LIN {X 0,Y 310.323,Z 1135.59,A -85,B 0,C 180,E1 15003.805,E2 15003.805} C_VEL
LIN {X 0,Y 314.17,Z 1124.911,A -85,B 0,C 180,E1 14999.811,E2 14999.811} C_VEL
LIN {X 0,Y 318.874,Z 1112.724,A -85,B 0,C 180,E1 14996.072,E2 14996.072} C_VEL
LIN {X 0,Y 324.647,Z 1098.598,A -85,B 0,C 180,E1 14992.424,E2 14992.424} C_VEL
LIN {X 0,Y 330.405,Z 1084.681,A -85,B 0,C 180,E1 14989.411,E2 14989.411} C_VEL
LIN {X 0,Y 337.548,Z 1067.241,A -85,B 0,C 180,E1 14986.238,E2 14986.238} C_VEL
LIN {X 0,Y 344.264,Z 1050.446,A -85,B 0,C 180,E1 14983.682,E2 14983.682} C_VEL
LIN {X 0,Y 351.205,Z 1031.927,A -85,B 0,C 180,E1 14981.337,E2 14981.337} C_VEL
LIN {X 0,Y 357.94,Z 1012.865,A -85,B 0,C 180,E1 14979.306,E2 14979.306} C_VEL
LIN {X 0,Y 364.39,Z 992.442,A -85,B 0,C 180,E1 14977.528,E2 14977.528} C_VEL
LIN {X 0,Y 370.322,Z 971.659,A -85,B 0,C 180,E1 14976.036,E2 14976.036} C_VEL
LIN {X 0,Y 375.316,Z 951.31,A -85,B 0,C 180,E1 14974.861,E2 14974.861} C_VEL
LIN {X 0,Y 380.154,Z 927.978,A -85,B 0,C 180,E1 14973.796,E2 14973.796} C_VEL
LIN {X 0,Y 383.734,Z 906.313,A -85,B 0,C 180,E1 14973.058,E2 14973.058} C_VEL
LIN {X 0,Y 386.535,Z 881.758,A -85,B 0,C 180,E1 14972.438,E2 14972.438} C_VEL
LIN {X 0,Y 398.711,Z 690.492,A -85,B 0,C 180,E1 14968.671,E2 14968.671} C_VEL
LIN {X 0,Y 400.761,Z 658.99,A -85,B 0,C 180,E1 14968.053,E2 14968.053} C_VEL
LIN {X 0,Y 392.49,Z 644.745,A -85,B 0,C 180,E1 14965.137,E2 14965.137} C_VEL
LIN {X 0,Y 385.004,Z 632.908,A -85,B 0,C 180,E1 14962.121,E2 14962.121} C_VEL
LIN {X 0,Y 380.759,Z 626.867,A -85,B 0,C 180,E1 14960.2,E2 14960.2} C_VEL
LIN {X 0,Y 377.272,Z 622.196,A -85,B 0,C 180,E1 14958.463,E2 14958.463} C_VEL
LIN {X 0,Y 373.463,Z 617.117,A -85,B 0,C 180,E1 14956.326,E2 14956.326} C_VEL
LIN {X 0,Y 370.02,Z 612.377,A -85,B 0,C 180,E1 14954.075,E2 14954.075} C_VEL
LIN {X 0,Y 366.537,Z 608.515,A -85,B 0,C 180,E1 14951.406,E2 14951.406} C_VEL
LIN {X 0,Y 365.354,Z 606.34,A -85,B 0,C 180,E1 14950.246,E2 14950.246} C_VEL
LIN {X 0,Y 362.118,Z 603.229,A -85,B 0,C 180,E1 14946.5,E2 14946.5} C_VEL
LIN {X 0,Y 361.007,Z 600.343,A -85,B 0,C 180,E1 14944.129,E2 14944.129} C_VEL
LIN {X 0,Y 360.416,Z 600.177,A -85,B 0,C 180,E1 14936.819,E2 14936.819} C_VEL
LIN {X 0,Y 361.128,Z 600.593,A -85,B 0,C 180,E1 14934.996,E2 14934.996} C_VEL
LIN {X 0,Y 363.051,Z 604.515,A -85,B 0,C 180,E1 14931.607,E2 14931.607} C_VEL
LIN {X 0,Y 365.657,Z 606.777,A -85,B 0,C 180,E1 14928.885,E2 14928.885} C_VEL
LIN {X 0,Y 368.284,Z 610.838,A -85,B 0,C 180,E1 14926.577,E2 14926.577} C_VEL
LIN {X 0,Y 370.242,Z 612.802,A -85,B 0,C 180,E1 14925.187,E2 14925.187} C_VEL
LIN {X 0,Y 373.699,Z 617.381,A -85,B 0,C 180,E1 14922.964,E2 14922.964} C_VEL
LIN {X 0,Y 378.892,Z 624.313,A -85,B 0,C 180,E1 14920.138,E2 14920.138} C_VEL
LIN {X 0,Y 383.061,Z 630.072,A -85,B 0,C 180,E1 14918.164,E2 14918.164} C_VEL
LIN {X 0,Y 388.835,Z 638.03,A -85,B 0,C 180,E1 14915.746,E2 14915.746} C_VEL
LIN {X 0,Y 397.734,Z 651.353,A -85,B 0,C 180,E1 14912.488,E2 14912.488} C_VEL
LIN {X 0,Y 400.67,Z 656.231,A -85,B 0,C 180,E1 14911.501,E2 14911.501} C_VEL
LIN {X 0,Y 387.914,Z 856.221,A -85,B 0,C 180,E1 14907.587,E2 14907.587} C_VEL
LIN {X 0,Y 385.767,Z 879.846,A -85,B 0,C 180,E1 14907.046,E2 14907.046} C_VEL
LIN {X 0,Y 382.642,Z 902.799,A -85,B 0,C 180,E1 14906.324,E2 14906.324} C_VEL
LIN {X 0,Y 378.824,Z 923.719,A -85,B 0,C 180,E1 14905.436,E2 14905.436} C_VEL
LIN {X 0,Y 373.938,Z 945.868,A -85,B 0,C 180,E1 14904.246,E2 14904.246} C_VEL
LIN {X 0,Y 368.881,Z 965.062,A -85,B 0,C 180,E1 14902.964,E2 14902.964} C_VEL
LIN {X 0,Y 362.451,Z 986.567,A -85,B 0,C 180,E1 14901.211,E2 14901.211} C_VEL
LIN {X 0,Y 356.513,Z 1004.243,A -85,B 0,C 180,E1 14899.468,E2 14899.468} C_VEL
LIN {X 0,Y 349.249,Z 1023.997,A -85,B 0,C 180,E1 14897.131,E2 14897.131} C_VEL
LIN {X 0,Y 342.731,Z 1040.527,A -85,B 0,C 180,E1 14894.793,E2 14894.793} C_VEL
LIN {X 0,Y 335.925,Z 1056.776,A -85,B 0,C 180,E1 14892.045,E2 14892.045} C_VEL
LIN {X 0,Y 329.503,Z 1071.829,A -85,B 0,C 180,E1 14889.029,E2 14889.029} C_VEL
LIN {X 0,Y 323.5,Z 1085.447,A -85,B 0,C 180,E1 14885.744,E2 14885.744} C_VEL
LIN {X 0,Y 318.06,Z 1098.198,A -85,B 0,C 180,E1 14882.092,E2 14882.092} C_VEL
LIN {X 0,Y 313.614,Z 1108.925,A -85,B 0,C 180,E1 14878.363,E2 14878.363} C_VEL
LIN {X 0,Y 309.706,Z 1119.272,A -85,B 0,C 180,E1 14873.986,E2 14873.986} C_VEL
LIN {X 0,Y 307.195,Z 1126.919,A -85,B 0,C 180,E1 14869.984,E2 14869.984} C_VEL
LIN {X 0,Y 305.468,Z 1133.25,A -85,B 0,C 180,E1 14865.765,E2 14865.765} C_VEL
LIN {X 0,Y 304.592,Z 1137.667,A -85,B 0,C 180,E1 14861.936,E2 14861.936} C_VEL
LIN {X 0,Y 304.117,Z 1141.074,A -85,B 0,C 180,E1 14857.747,E2 14857.747} C_VEL
LIN {X 0,Y 303.996,Z 1142.818,A -85,B 0,C 180,E1 14854.15,E2 14854.15} C_VEL
LIN {X 0,Y 303.963,Z 1143.581,A -85,B 0,C 180,E1 14850.326,E2 14850.326} C_VEL
LIN {X 0,Y 303.98,Z 1142.983,A -85,B 0,C 180,E1 14846.229,E2 14846.229} C_VEL
LIN {X 0,Y 304.085,Z 1141.349,A -85,B 0,C 180,E1 14842.633,E2 14842.633} C_VEL
LIN {X 0,Y 304.486,Z 1138.367,A -85,B 0,C 180,E1 14838.637,E2 14838.637} C_VEL
LIN {X 0,Y 305.382,Z 1133.619,A -85,B 0,C 180,E1 14834.427,E2 14834.427} C_VEL
LIN {X 0,Y 305.467,Z 1133.26,A -85,B 0,C 180,E1 14834.147,E2 14834.147} C_VEL
LIN {X 0,Y 304.971,Z 1131.474,A -85,B 0,C 180,E1 14832.733,E2 14832.733} C_VEL
LIN {X 0,Y 300.512,Z 1126.313,A -85,B 0,C 180,E1 14828.918,E2 14828.918} C_VEL
LIN {X 0,Y 300.483,Z 1124.298,A -85,B 0,C 180,E1 14827.7,E2 14827.7} C_VEL
LIN {X 0,Y 303.77,Z 1115.533,A -85,B 0,C 180,E1 14823.408,E2 14823.408} C_VEL
LIN {X 0,Y 307.804,Z 1105.953,A -85,B 0,C 180,E1 14819.553,E2 14819.553} C_VEL
LIN {X 0,Y 312.855,Z 1094.529,A -85,B 0,C 180,E1 14815.773,E2 14815.773} C_VEL
LIN {X 0,Y 318.735,Z 1081.794,A -85,B 0,C 180,E1 14812.234,E2 14812.234} C_VEL
LIN {X 0,Y 325.377,Z 1067.137,A -85,B 0,C 180,E1 14808.883,E2 14808.883} C_VEL
LIN {X 0,Y 332.647,Z 1050.932,A -85,B 0,C 180,E1 14805.786,E2 14805.786} C_VEL
LIN {X 0,Y 339.306,Z 1035.304,A -85,B 0,C 180,E1 14803.293,E2 14803.293} C_VEL
LIN {X 0,Y 347.012,Z 1016.058,A -85,B 0,C 180,E1 14800.73,E2 14800.73} C_VEL
LIN {X 0,Y 353.723,Z 997.925,A -85,B 0,C 180,E1 14798.725,E2 14798.725} C_VEL
LIN {X 0,Y 360.235,Z 978.29,A -85,B 0,C 180,E1 14796.931,E2 14796.931} C_VEL
LIN {X 0,Y 366.199,Z 958.243,A -85,B 0,C 180,E1 14795.411,E2 14795.411} C_VEL
LIN {X 0,Y 371.457,Z 937.38,A -85,B 0,C 180,E1 14794.136,E2 14794.136} C_VEL
LIN {X 0,Y 376.2,Z 915.233,A -85,B 0,C 180,E1 14793.049,E2 14793.049} C_VEL
LIN {X 0,Y 379.82,Z 893.219,A -85,B 0,C 180,E1 14792.229,E2 14792.229} C_VEL
LIN {X 0,Y 382.736,Z 869.272,A -85,B 0,C 180,E1 14791.578,E2 14791.578} C_VEL
LIN {X 0,Y 394.662,Z 690.82,A -85,B 0,C 180,E1 14788.052,E2 14788.052} C_VEL
LIN {X 0,Y 396.631,Z 660.49,A -85,B 0,C 180,E1 14787.432,E2 14787.432} C_VEL
LIN {X 0,Y 388.655,Z 648.175,A -85,B 0,C 180,E1 14784.509,E2 14784.509} C_VEL
LIN {X 0,Y 382.448,Z 639.194,A -85,B 0,C 180,E1 14781.913,E2 14781.913} C_VEL
LIN {X 0,Y 378.405,Z 633.571,A -85,B 0,C 180,E1 14780.01,E2 14780.01} C_VEL
LIN {X 0,Y 375.594,Z 629.676,A -85,B 0,C 180,E1 14778.549,E2 14778.549} C_VEL
LIN {X 0,Y 371.88,Z 624.709,A -85,B 0,C 180,E1 14776.398,E2 14776.398} C_VEL
LIN {X 0,Y 368.336,Z 619.786,A -85,B 0,C 180,E1 14773.981,E2 14773.981} C_VEL
LIN {X 0,Y 365.292,Z 616.25,A -85,B 0,C 180,E1 14771.526,E2 14771.526} C_VEL
LIN {X 0,Y 364.226,Z 614.277,A -85,B 0,C 180,E1 14770.439,E2 14770.439} C_VEL
LIN {X 0,Y 361.038,Z 611.018,A -85,B 0,C 180,E1 14766.52,E2 14766.52} C_VEL
LIN {X 0,Y 360.042,Z 608.276,A -85,B 0,C 180,E1 14764.141,E2 14764.141} C_VEL
LIN {X 0,Y 360.043,Z 608.283,A -85,B 0,C 180,E1 14756.338,E2 14756.338} C_VEL
LIN {X 0,Y 362.332,Z 612.803,A -85,B 0,C 180,E1 14752.07,E2 14752.07} C_VEL
LIN {X 0,Y 364.46,Z 614.581,A -85,B 0,C 180,E1 14749.808,E2 14749.808} C_VEL
LIN {X 0,Y 367.19,Z 618.789,A -85,B 0,C 180,E1 14747.338,E2 14747.338} C_VEL
LIN {X 0,Y 368.856,Z 620.49,A -85,B 0,C 180,E1 14746.12,E2 14746.12} C_VEL
LIN {X 0,Y 372.39,Z 625.157,A -85,B 0,C 180,E1 14743.786,E2 14743.786} C_VEL
LIN {X 0,Y 377.467,Z 632.272,A -85,B 0,C 180,E1 14740.946,E2 14740.946} C_VEL
LIN {X 0,Y 381.184,Z 637.463,A -85,B 0,C 180,E1 14739.141,E2 14739.141} C_VEL
LIN {X 0,Y 385.902,Z 644.86,A -85,B 0,C 180,E1 14737.05,E2 14737.05} C_VEL
LIN {X 0,Y 391.999,Z 654.977,A -85,B 0,C 180,E1 14734.627,E2 14734.627} C_VEL
LIN {X 0,Y 396.821,Z 663.696,A -85,B 0,C 180,E1 14732.874,E2 14732.874} C_VEL
LIN {X 0,Y 382.995,Z 873.743,A -85,B 0,C 180,E1 14728.753,E2 14728.753} C_VEL
LIN {X 0,Y 380.728,Z 896.852,A -85,B 0,C 180,E1 14728.218,E2 14728.218} C_VEL
LIN {X 0,Y 376.911,Z 921.624,A -85,B 0,C 180,E1 14727.459,E2 14727.459} C_VEL
LIN {X 0,Y 372.941,Z 941.713,A -85,B 0,C 180,E1 14726.63,E2 14726.63} C_VEL
LIN {X 0,Y 367.489,Z 964.391,A -85,B 0,C 180,E1 14725.43,E2 14725.43} C_VEL
LIN {X 0,Y 361.774,Z 984.881,A -85,B 0,C 180,E1 14724.075,E2 14724.075} C_VEL
LIN {X 0,Y 355.238,Z 1005.335,A -85,B 0,C 180,E1 14722.402,E2 14722.402} C_VEL
LIN {X 0,Y 348.52,Z 1024.568,A -85,B 0,C 180,E1 14720.509,E2 14720.509} C_VEL
LIN {X 0,Y 341.201,Z 1043.572,A -85,B 0,C 180,E1 14718.227,E2 14718.227} C_VEL
LIN {X 0,Y 333.849,Z 1061.702,A -85,B 0,C 180,E1 14715.622,E2 14715.622} C_VEL
LIN {X 0,Y 327.017,Z 1077.671,A -85,B 0,C 180,E1 14712.867,E2 14712.867} C_VEL
LIN {X 0,Y 319.73,Z 1094.407,A -85,B 0,C 180,E1 14709.406,E2 14709.406} C_VEL
LIN {X 0,Y 313.658,Z 1108.501,A -85,B 0,C 180,E1 14705.912,E2 14705.912} C_VEL
LIN {X 0,Y 308.33,Z 1121.103,A -85,B 0,C 180,E1 14702.128,E2 14702.128} C_VEL
LIN {X 0,Y 303.91,Z 1132.469,A -85,B 0,C 180,E1 14698.064,E2 14698.064} C_VEL
LIN {X 0,Y 300.611,Z 1141.876,A -85,B 0,C 180,E1 14693.94,E2 14693.94} C_VEL
LIN {X 0,Y 298.166,Z 1150.31,A -85,B 0,C 180,E1 14689.389,E2 14689.389} C_VEL
LIN {X 0,Y 296.881,Z 1156.088,A -85,B 0,C 180,E1 14685.43,E2 14685.43} C_VEL
LIN {X 0,Y 296.169,Z 1161.086,A -85,B 0,C 180,E1 14680.897,E2 14680.897} C_VEL
LIN {X 0,Y 295.965,Z 1163.871,A -85,B 0,C 180,E1 14677.18,E2 14677.18} C_VEL
LIN {X 0,Y 295.95,Z 1165.555,A -85,B 0,C 180,E1 14673.486,E2 14673.486} C_VEL
LIN {X 0,Y 295.962,Z 1166.074,A -85,B 0,C 180,E1 14669.59,E2 14669.59} C_VEL
LIN {X 0,Y 295.962,Z 1165.342,A -85,B 0,C 180,E1 14665.931,E2 14665.931} C_VEL
LIN {X 0,Y 295.992,Z 1163.512,A -85,B 0,C 180,E1 14662.234,E2 14662.234} C_VEL
LIN {X 0,Y 296.296,Z 1159.96,A -85,B 0,C 180,E1 14657.923,E2 14657.923} C_VEL
LIN {X 0,Y 297.034,Z 1155.291,A -85,B 0,C 180,E1 14653.976,E2 14653.976} C_VEL
LIN {X 0,Y 298.61,Z 1148.673,A -85,B 0,C 180,E1 14649.62,E2 14649.62} C_VEL
LIN {X 0,Y 301.021,Z 1140.61,A -85,B 0,C 180,E1 14645.468,E2 14645.468} C_VEL
LIN {X 0,Y 304.663,Z 1130.418,A -85,B 0,C 180,E1 14641.155,E2 14641.155} C_VEL
LIN {X 0,Y 309.058,Z 1119.318,A -85,B 0,C 180,E1 14637.297,E2 14637.297} C_VEL
LIN {X 0,Y 314.85,Z 1105.605,A -85,B 0,C 180,E1 14633.342,E2 14633.342} C_VEL
LIN {X 0,Y 321.144,Z 1091.219,A -85,B 0,C 180,E1 14629.872,E2 14629.872} C_VEL
LIN {X 0,Y 328.027,Z 1075.258,A -85,B 0,C 180,E1 14626.699,E2 14626.699} C_VEL
LIN {X 0,Y 335.328,Z 1058.003,A -85,B 0,C 180,E1 14623.814,E2 14623.814} C_VEL
LIN {X 0,Y 342.149,Z 1041.054,A -85,B 0,C 180,E1 14621.455,E2 14621.455} C_VEL
LIN {X 0,Y 349.556,Z 1021.471,A -85,B 0,C 180,E1 14619.179,E2 14619.179} C_VEL
LIN {X 0,Y 356.069,Z 1002.737,A -85,B 0,C 180,E1 14617.374,E2 14617.374} C_VEL
LIN {X 0,Y 362.647,Z 981.642,A -85,B 0,C 180,E1 14615.706,E2 14615.706} C_VEL
LIN {X 0,Y 368.003,Z 962.244,A -85,B 0,C 180,E1 14614.45,E2 14614.45} C_VEL
LIN {X 0,Y 373.241,Z 939.947,A -85,B 0,C 180,E1 14613.299,E2 14613.299} C_VEL
LIN {X 0,Y 377.27,Z 919.347,A -85,B 0,C 180,E1 14612.467,E2 14612.467} C_VEL
LIN {X 0,Y 380.769,Z 895.853,A -85,B 0,C 180,E1 14611.764,E2 14611.764} C_VEL
LIN {X 0,Y 383.036,Z 872.053,A -85,B 0,C 180,E1 14611.22,E2 14611.22} C_VEL
LIN {X 0,Y 396.739,Z 663.465,A -85,B 0,C 180,E1 14607.129,E2 14607.129} C_VEL
LIN {X 0,Y 389.401,Z 650.607,A -85,B 0,C 180,E1 14604.418,E2 14604.418} C_VEL
LIN {X 0,Y 382.164,Z 638.896,A -85,B 0,C 180,E1 14601.365,E2 14601.365} C_VEL
LIN {X 0,Y 378.422,Z 633.662,A -85,B 0,C 180,E1 14599.606,E2 14599.606} C_VEL
LIN {X 0,Y 375.456,Z 629.581,A -85,B 0,C 180,E1 14598.074,E2 14598.074} C_VEL
LIN {X 0,Y 371.864,Z 624.679,A -85,B 0,C 180,E1 14595.997,E2 14595.997} C_VEL
LIN {X 0,Y 368.174,Z 619.697,A -85,B 0,C 180,E1 14593.506,E2 14593.506} C_VEL
LIN {X 0,Y 365.049,Z 615.916,A -85,B 0,C 180,E1 14590.973,E2 14590.973} C_VEL
LIN {X 0,Y 364.052,Z 614.127,A -85,B 0,C 180,E1 14589.963,E2 14589.963} C_VEL
LIN {X 0,Y 360.855,Z 610.766,A -85,B 0,C 180,E1 14586.044,E2 14586.044} C_VEL
LIN {X 0,Y 359.96,Z 608.269,A -85,B 0,C 180,E1 14583.982,E2 14583.982} C_VEL
LIN {X 0,Y 359.498,Z 608.138,A -85,B 0,C 180,E1 14576.633,E2 14576.633} C_VEL
LIN {X 0,Y 360.078,Z 608.513,A -85,B 0,C 180,E1 14575.141,E2 14575.141} C_VEL
LIN {X 0,Y 361.954,Z 612.395,A -85,B 0,C 180,E1 14571.741,E2 14571.741} C_VEL
LIN {X 0,Y 364.428,Z 614.657,A -85,B 0,C 180,E1 14569.087,E2 14569.087} C_VEL
LIN {X 0,Y 367.013,Z 618.639,A -85,B 0,C 180,E1 14566.771,E2 14566.771} C_VEL
LIN {X 0,Y 368.791,Z 620.478,A -85,B 0,C 180,E1 14565.476,E2 14565.476} C_VEL
LIN {X 0,Y 372.223,Z 625.071,A -85,B 0,C 180,E1 14563.216,E2 14563.216} C_VEL
LIN {X 0,Y 377.185,Z 631.895,A -85,B 0,C 180,E1 14560.447,E2 14560.447} C_VEL
LIN {X 0,Y 381.204,Z 637.558,A -85,B 0,C 180,E1 14558.497,E2 14558.497} C_VEL
LIN {X 0,Y 386.708,Z 645.323,A -85,B 0,C 180,E1 14556.131,E2 14556.131} C_VEL
LIN {X 0,Y 395.16,Z 658.231,A -85,B 0,C 180,E1 14552.95,E2 14552.95} C_VEL
LIN {X 0,Y 396.616,Z 660.877,A -85,B 0,C 180,E1 14552.433,E2 14552.433} C_VEL
LIN {X 0,Y 383.418,Z 860.114,A -85,B 0,C 180,E1 14548.521,E2 14548.521} C_VEL
LIN {X 0,Y 381.23,Z 882.282,A -85,B 0,C 180,E1 14547.997,E2 14547.997} C_VEL
LIN {X 0,Y 377.759,Z 905.918,A -85,B 0,C 180,E1 14547.224,E2 14547.224} C_VEL
LIN {X 0,Y 373.897,Z 926.162,A -85,B 0,C 180,E1 14546.347,E2 14546.347} C_VEL
LIN {X 0,Y 368.699,Z 948.424,A -85,B 0,C 180,E1 14545.119,E2 14545.119} C_VEL
LIN {X 0,Y 363.509,Z 967.365,A -85,B 0,C 180,E1 14543.833,E2 14543.833} C_VEL
LIN {X 0,Y 357.121,Z 987.761,A -85,B 0,C 180,E1 14542.143,E2 14542.143} C_VEL
LIN {X 0,Y 350.732,Z 1006.09,A -85,B 0,C 180,E1 14540.314,E2 14540.314} C_VEL
LIN {X 0,Y 343.482,Z 1024.939,A -85,B 0,C 180,E1 14538.046,E2 14538.046} C_VEL
LIN {X 0,Y 336.512,Z 1041.934,A -85,B 0,C 180,E1 14535.61,E2 14535.61} C_VEL
LIN {X 0,Y 329.446,Z 1058,A -85,B 0,C 180,E1 14532.832,E2 14532.832} C_VEL
LIN {X 0,Y 322.577,Z 1073.326,A -85,B 0,C 180,E1 14529.682,E2 14529.682} C_VEL
LIN {X 0,Y 316.51,Z 1086.447,A -85,B 0,C 180,E1 14526.435,E2 14526.435} C_VEL
LIN {X 0,Y 310.555,Z 1099.631,A -85,B 0,C 180,E1 14522.526,E2 14522.526} C_VEL
LIN {X 0,Y 306.154,Z 1109.739,A -85,B 0,C 180,E1 14518.905,E2 14518.905} C_VEL
LIN {X 0,Y 302.201,Z 1119.55,A -85,B 0,C 180,E1 14514.639,E2 14514.639} C_VEL
LIN {X 0,Y 299.495,Z 1127.228,A -85,B 0,C 180,E1 14510.521,E2 14510.521} C_VEL
LIN {X 0,Y 297.582,Z 1133.714,A -85,B 0,C 180,E1 14506.065,E2 14506.065} C_VEL
LIN {X 0,Y 296.599,Z 1138.371,A -85,B 0,C 180,E1 14501.867,E2 14501.867} C_VEL
LIN {X 0,Y 296.112,Z 1141.595,A -85,B 0,C 180,E1 14497.568,E2 14497.568} C_VEL
LIN {X 0,Y 295.995,Z 1143.249,A -85,B 0,C 180,E1 14493.874,E2 14493.874} C_VEL
LIN {X 0,Y 295.973,Z 1143.908,A -85,B 0,C 180,E1 14489.807,E2 14489.807} C_VEL
LIN {X 0,Y 296.002,Z 1143.152,A -85,B 0,C 180,E1 14485.739,E2 14485.739} C_VEL
LIN {X 0,Y 296.158,Z 1141.323,A -85,B 0,C 180,E1 14481.849,E2 14481.849} C_VEL
LIN {X 0,Y 296.71,Z 1137.672,A -85,B 0,C 180,E1 14477.348,E2 14477.348} C_VEL
LIN {X 0,Y 297.806,Z 1132.941,A -85,B 0,C 180,E1 14473.218,E2 14473.218} C_VEL
LIN {X 0,Y 299.892,Z 1126.025,A -85,B 0,C 180,E1 14468.69,E2 14468.69} C_VEL
LIN {X 0,Y 300.483,Z 1124.298,A -85,B 0,C 180,E1 14467.7,E2 14467.7} C_VEL
LIN {X 0,Y 300.434,Z 1121.89,A -85,B 0,C 180,E1 14466.293,E2 14466.293} C_VEL
LIN {X 0,Y 297.378,Z 1115.16,A -85,B 0,C 180,E1 14462.471,E2 14462.471} C_VEL
LIN {X 0,Y 297.827,Z 1112.655,A -85,B 0,C 180,E1 14461.283,E2 14461.283} C_VEL
LIN {X 0,Y 302.7,Z 1101.884,A -85,B 0,C 180,E1 14457.2,E2 14457.2} C_VEL
LIN {X 0,Y 308.496,Z 1089.823,A -85,B 0,C 180,E1 14453.391,E2 14453.391} C_VEL
LIN {X 0,Y 315.005,Z 1076.254,A -85,B 0,C 180,E1 14449.884,E2 14449.884} C_VEL
LIN {X 0,Y 322.472,Z 1060.543,A -85,B 0,C 180,E1 14446.502,E2 14446.502} C_VEL
LIN {X 0,Y 329.497,Z 1045.241,A -85,B 0,C 180,E1 14443.763,E2 14443.763} C_VEL
LIN {X 0,Y 337.167,Z 1027.551,A -85,B 0,C 180,E1 14441.129,E2 14441.129} C_VEL
LIN {X 0,Y 344.124,Z 1010.415,A -85,B 0,C 180,E1 14438.993,E2 14438.993} C_VEL
LIN {X 0,Y 351.191,Z 991.173,A -85,B 0,C 180,E1 14437.004,E2 14437.004} C_VEL
LIN {X 0,Y 357.477,Z 972.322,A -85,B 0,C 180,E1 14435.379,E2 14435.379} C_VEL
LIN {X 0,Y 363.46,Z 951.595,A -85,B 0,C 180,E1 14433.921,E2 14433.921} C_VEL
LIN {X 0,Y 368.561,Z 931.288,A -85,B 0,C 180,E1 14432.755,E2 14432.755} C_VEL
LIN {X 0,Y 372.973,Z 909.487,A -85,B 0,C 180,E1 14431.773,E2 14431.773} C_VEL
LIN {X 0,Y 376.463,Z 888.081,A -85,B 0,C 180,E1 14431.026,E2 14431.026} C_VEL
LIN {X 0,Y 378.998,Z 864.998,A -85,B 0,C 180,E1 14430.448,E2 14430.448} C_VEL
LIN {X 0,Y 392.66,Z 667.126,A -85,B 0,C 180,E1 14426.551,E2 14426.551} C_VEL
LIN {X 0,Y 392.75,Z 665.236,A -85,B 0,C 180,E1 14426.501,E2 14426.501} C_VEL
LIN {X 0,Y 384.149,Z 651.782,A -85,B 0,C 180,E1 14423.143,E2 14423.143} C_VEL
LIN {X 0,Y 377.425,Z 642.064,A -85,B 0,C 180,E1 14420.064,E2 14420.064} C_VEL
LIN {X 0,Y 373.665,Z 636.906,A -85,B 0,C 180,E1 14418.083,E2 14418.083} C_VEL
LIN {X 0,Y 370.3,Z 632.269,A -85,B 0,C 180,E1 14416.067,E2 14416.067} C_VEL
LIN {X 0,Y 366.734,Z 627.329,A -85,B 0,C 180,E1 14413.561,E2 14413.561} C_VEL
LIN {X 0,Y 363.749,Z 623.51,A -85,B 0,C 180,E1 14411.014,E2 14411.014} C_VEL
LIN {X 0,Y 362.935,Z 622.069,A -85,B 0,C 180,E1 14410.156,E2 14410.156} C_VEL
LIN {X 0,Y 359.883,Z 618.731,A -85,B 0,C 180,E1 14406.221,E2 14406.221} C_VEL
LIN {X 0,Y 359.005,Z 616.202,A -85,B 0,C 180,E1 14403.993,E2 14403.993} C_VEL
LIN {X 0,Y 359.07,Z 616.224,A -85,B 0,C 180,E1 14396.328,E2 14396.328} C_VEL
LIN {X 0,Y 360.991,Z 620.417,A -85,B 0,C 180,E1 14392.52,E2 14392.52} C_VEL
LIN {X 0,Y 363.241,Z 622.444,A -85,B 0,C 180,E1 14390.014,E2 14390.014} C_VEL
LIN {X 0,Y 365.923,Z 626.589,A -85,B 0,C 180,E1 14387.534,E2 14387.534} C_VEL
LIN {X 0,Y 367.549,Z 628.4,A -85,B 0,C 180,E1 14386.31,E2 14386.31} C_VEL
LIN {X 0,Y 371.506,Z 633.867,A -85,B 0,C 180,E1 14383.666,E2 14383.666} C_VEL
LIN {X 0,Y 375.63,Z 639.633,A -85,B 0,C 180,E1 14381.332,E2 14381.332} C_VEL
LIN {X 0,Y 379.571,Z 645.276,A -85,B 0,C 180,E1 14379.371,E2 14379.371} C_VEL
LIN {X 0,Y 384.969,Z 653.991,A -85,B 0,C 180,E1 14376.95,E2 14376.95} C_VEL
LIN {X 0,Y 391.59,Z 665.539,A -85,B 0,C 180,E1 14374.315,E2 14374.315} C_VEL
LIN {X 0,Y 392.874,Z 668.184,A -85,B 0,C 180,E1 14373.826,E2 14373.826} C_VEL
LIN {X 0,Y 378.717,Z 875.394,A -85,B 0,C 180,E1 14369.752,E2 14369.752} C_VEL
LIN {X 0,Y 376.41,Z 897.705,A -85,B 0,C 180,E1 14369.23,E2 14369.23} C_VEL
LIN {X 0,Y 372.481,Z 922.139,A -85,B 0,C 180,E1 14368.475,E2 14368.475} C_VEL
LIN {X 0,Y 368.231,Z 942.906,A -85,B 0,C 180,E1 14367.614,E2 14367.614} C_VEL
LIN {X 0,Y 362.847,Z 964.426,A -85,B 0,C 180,E1 14366.467,E2 14366.467} C_VEL
LIN {X 0,Y 357.046,Z 984.581,A -85,B 0,C 180,E1 14365.136,E2 14365.136} C_VEL
LIN {X 0,Y 350.214,Z 1005.252,A -85,B 0,C 180,E1 14363.446,E2 14363.446} C_VEL
LIN {X 0,Y 343.072,Z 1024.958,A -85,B 0,C 180,E1 14361.497,E2 14361.497} C_VEL
LIN {X 0,Y 335.478,Z 1043.88,A -85,B 0,C 180,E1 14359.202,E2 14359.202} C_VEL
LIN {X 0,Y 327.54,Z 1062.576,A -85,B 0,C 180,E1 14356.469,E2 14356.469} C_VEL
LIN {X 0,Y 320.526,Z 1078.3,A -85,B 0,C 180,E1 14353.705,E2 14353.705} C_VEL
LIN {X 0,Y 313.292,Z 1094.094,A -85,B 0,C 180,E1 14350.381,E2 14350.381} C_VEL
LIN {X 0,Y 306.905,Z 1108.188,A -85,B 0,C 180,E1 14346.83,E2 14346.83} C_VEL
LIN {X 0,Y 301.256,Z 1120.79,A -85,B 0,C 180,E1 14342.977,E2 14342.977} C_VEL
LIN {X 0,Y 296.551,Z 1132.156,A -85,B 0,C 180,E1 14338.825,E2 14338.825} C_VEL
LIN {X 0,Y 293.017,Z 1141.565,A -85,B 0,C 180,E1 14334.601,E2 14334.601} C_VEL
LIN {X 0,Y 290.379,Z 1150.001,A -85,B 0,C 180,E1 14329.93,E2 14329.93} C_VEL
LIN {X 0,Y 288.981,Z 1155.781,A -85,B 0,C 180,E1 14325.862,E2 14325.862} C_VEL
LIN {X 0,Y 288.202,Z 1160.782,A -85,B 0,C 180,E1 14321.202,E2 14321.202} C_VEL
LIN {X 0,Y 287.97,Z 1163.569,A -85,B 0,C 180,E1 14317.381,E2 14317.381} C_VEL
LIN {X 0,Y 287.956,Z 1165.255,A -85,B 0,C 180,E1 14313.583,E2 14313.583} C_VEL
LIN {X 0,Y 287.966,Z 1165.766,A -85,B 0,C 180,E1 14309.509,E2 14309.509} C_VEL
LIN {X 0,Y 287.966,Z 1164.97,A -85,B 0,C 180,E1 14305.619,E2 14305.619} C_VEL
LIN {X 0,Y 288.021,Z 1163.091,A -85,B 0,C 180,E1 14301.817,E2 14301.817} C_VEL
LIN {X 0,Y 288.364,Z 1159.441,A -85,B 0,C 180,E1 14297.382,E2 14297.382} C_VEL
LIN {X 0,Y 289.228,Z 1154.624,A -85,B 0,C 180,E1 14293.251,E2 14293.251} C_VEL
LIN {X 0,Y 291.159,Z 1147.27,A -85,B 0,C 180,E1 14288.441,E2 14288.441} C_VEL
LIN {X 0,Y 293.755,Z 1139.463,A -85,B 0,C 180,E1 14284.388,E2 14284.388} C_VEL
LIN {X 0,Y 297.766,Z 1129.048,A -85,B 0,C 180,E1 14279.978,E2 14279.978} C_VEL
LIN {X 0,Y 302.582,Z 1117.795,A -85,B 0,C 180,E1 14276.037,E2 14276.037} C_VEL
LIN {X 0,Y 308.469,Z 1104.573,A -85,B 0,C 180,E1 14272.22,E2 14272.22} C_VEL
LIN {X 0,Y 315.161,Z 1090.063,A -85,B 0,C 180,E1 14268.708,E2 14268.708} C_VEL
LIN {X 0,Y 322.204,Z 1074.472,A -85,B 0,C 180,E1 14265.591,E2 14265.591} C_VEL
LIN {X 0,Y 330.086,Z 1056.563,A -85,B 0,C 180,E1 14262.602,E2 14262.602} C_VEL
LIN {X 0,Y 337.079,Z 1039.888,A -85,B 0,C 180,E1 14260.288,E2 14260.288} C_VEL
LIN {X 0,Y 344.682,Z 1020.416,A -85,B 0,C 180,E1 14258.04,E2 14258.04} C_VEL
LIN {X 0,Y 351.152,Z 1002.425,A -85,B 0,C 180,E1 14256.311,E2 14256.311} C_VEL
LIN {X 0,Y 357.935,Z 981.358,A -85,B 0,C 180,E1 14254.647,E2 14254.647} C_VEL
LIN {X 0,Y 363.604,Z 961.44,A -85,B 0,C 180,E1 14253.364,E2 14253.364} C_VEL
LIN {X 0,Y 368.859,Z 939.635,A -85,B 0,C 180,E1 14252.248,E2 14252.248} C_VEL
LIN {X 0,Y 372.94,Z 919.361,A -85,B 0,C 180,E1 14251.434,E2 14251.434} C_VEL
LIN {X 0,Y 376.574,Z 895.699,A -85,B 0,C 180,E1 14250.727,E2 14250.727} C_VEL
LIN {X 0,Y 378.909,Z 871.983,A -85,B 0,C 180,E1 14250.184,E2 14250.184} C_VEL
LIN {X 0,Y 392.788,Z 667.957,A -85,B 0,C 180,E1 14246.177,E2 14246.177} C_VEL
LIN {X 0,Y 386.541,Z 656.796,A -85,B 0,C 180,E1 14243.758,E2 14243.758} C_VEL
LIN {X 0,Y 379.99,Z 645.93,A -85,B 0,C 180,E1 14240.887,E2 14240.887} C_VEL
LIN {X 0,Y 376.129,Z 640.435,A -85,B 0,C 180,E1 14239.004,E2 14239.004} C_VEL
LIN {X 0,Y 373.523,Z 636.805,A -85,B 0,C 180,E1 14237.606,E2 14237.606} C_VEL
LIN {X 0,Y 370.155,Z 632.107,A -85,B 0,C 180,E1 14235.591,E2 14235.591} C_VEL
LIN {X 0,Y 366.781,Z 627.408,A -85,B 0,C 180,E1 14233.237,E2 14233.237} C_VEL
LIN {X 0,Y 363.659,Z 623.461,A -85,B 0,C 180,E1 14230.615,E2 14230.615} C_VEL
LIN {X 0,Y 362.76,Z 621.909,A -85,B 0,C 180,E1 14229.679,E2 14229.679} C_VEL
LIN {X 0,Y 359.699,Z 618.474,A -85,B 0,C 180,E1 14225.743,E2 14225.743} C_VEL
LIN {X 0,Y 358.916,Z 616.194,A -85,B 0,C 180,E1 14223.833,E2 14223.833} C_VEL
LIN {X 0,Y 358.524,Z 616.079,A -85,B 0,C 180,E1 14216.625,E2 14216.625} C_VEL
LIN {X 0,Y 359.031,Z 616.429,A -85,B 0,C 180,E1 14215.287,E2 14215.287} C_VEL
LIN {X 0,Y 360.859,Z 620.274,A -85,B 0,C 180,E1 14211.876,E2 14211.876} C_VEL
LIN {X 0,Y 363.134,Z 622.366,A -85,B 0,C 180,E1 14209.369,E2 14209.369} C_VEL
LIN {X 0,Y 365.846,Z 626.54,A -85,B 0,C 180,E1 14206.889,E2 14206.889} C_VEL
LIN {X 0,Y 367.384,Z 628.213,A -85,B 0,C 180,E1 14205.741,E2 14205.741} C_VEL
LIN {X 0,Y 371.592,Z 634.097,A -85,B 0,C 180,E1 14202.945,E2 14202.945} C_VEL
LIN {X 0,Y 375.489,Z 639.472,A -85,B 0,C 180,E1 14200.76,E2 14200.76} C_VEL
LIN {X 0,Y 379.437,Z 645.153,A -85,B 0,C 180,E1 14198.797,E2 14198.797} C_VEL
LIN {X 0,Y 384.848,Z 653.017,A -85,B 0,C 180,E1 14196.415,E2 14196.415} C_VEL
LIN {X 0,Y 392.684,Z 665.231,A -85,B 0,C 180,E1 14193.391,E2 14193.391} C_VEL
LIN {X 0,Y 379.342,Z 859.968,A -85,B 0,C 180,E1 14189.562,E2 14189.562} C_VEL
LIN {X 0,Y 377.083,Z 882.308,A -85,B 0,C 180,E1 14189.036,E2 14189.036} C_VEL
LIN {X 0,Y 373.477,Z 906.23,A -85,B 0,C 180,E1 14188.258,E2 14188.258} C_VEL
LIN {X 0,Y 369.546,Z 926.262,A -85,B 0,C 180,E1 14187.395,E2 14187.395} C_VEL
LIN {X 0,Y 364.118,Z 948.845,A -85,B 0,C 180,E1 14186.153,E2 14186.153} C_VEL
LIN {X 0,Y 358.508,Z 968.672,A -85,B 0,C 180,E1 14184.803,E2 14184.803} C_VEL
LIN {X 0,Y 351.917,Z 988.875,A -85,B 0,C 180,E1 14183.111,E2 14183.111} C_VEL
LIN {X 0,Y 345.09,Z 1007.772,A -85,B 0,C 180,E1 14181.206,E2 14181.206} C_VEL
LIN {X 0,Y 337.832,Z 1025.82,A -85,B 0,C 180,E1 14179.001,E2 14179.001} C_VEL
LIN {X 0,Y 330.595,Z 1042.787,A -85,B 0,C 180,E1 14176.541,E2 14176.541} C_VEL
LIN {X 0,Y 323.032,Z 1059.224,A -85,B 0,C 180,E1 14173.65,E2 14173.65} C_VEL
LIN {X 0,Y 315.884,Z 1074.396,A -85,B 0,C 180,E1 14170.458,E2 14170.458} C_VEL
LIN {X 0,Y 309.569,Z 1087.447,A -85,B 0,C 180,E1 14167.156,E2 14167.156} C_VEL
LIN {X 0,Y 303.282,Z 1100.62,A -85,B 0,C 180,E1 14163.134,E2 14163.134} C_VEL
LIN {X 0,Y 298.299,Z 1111.559,A -85,B 0,C 180,E1 14159.08,E2 14159.08} C_VEL
LIN {X 0,Y 294.399,Z 1120.648,A -85,B 0,C 180,E1 14154.907,E2 14154.907} C_VEL
LIN {X 0,Y 291.484,Z 1128.537,A -85,B 0,C 180,E1 14150.481,E2 14150.481} C_VEL
LIN {X 0,Y 289.587,Z 1134.601,A -85,B 0,C 180,E1 14146.035,E2 14146.035} C_VEL
LIN {X 0,Y 288.567,Z 1139.219,A -85,B 0,C 180,E1 14141.594,E2 14141.594} C_VEL
LIN {X 0,Y 288.122,Z 1142.006,A -85,B 0,C 180,E1 14137.578,E2 14137.578} C_VEL
LIN {X 0,Y 287.997,Z 1143.616,A -85,B 0,C 180,E1 14133.783,E2 14133.783} C_VEL
LIN {X 0,Y 287.97,Z 1144.178,A -85,B 0,C 180,E1 14129.538,E2 14129.538} C_VEL
LIN {X 0,Y 288.01,Z 1143.452,A -85,B 0,C 180,E1 14125.62,E2 14125.62} C_VEL
LIN {X 0,Y 288.194,Z 1141.625,A -85,B 0,C 180,E1 14121.622,E2 14121.622} C_VEL
LIN {X 0,Y 288.793,Z 1137.976,A -85,B 0,C 180,E1 14116.995,E2 14116.995} C_VEL
LIN {X 0,Y 289.991,Z 1133.246,A -85,B 0,C 180,E1 14112.752,E2 14112.752} C_VEL
LIN {X 0,Y 292.246,Z 1126.332,A -85,B 0,C 180,E1 14108.104,E2 14108.104} C_VEL
LIN {X 0,Y 295.517,Z 1118.071,A -85,B 0,C 180,E1 14103.69,E2 14103.69} C_VEL
LIN {X 0,Y 297.827,Z 1112.655,A -85,B 0,C 180,E1 14101.283,E2 14101.283} C_VEL
LIN {X 0,Y 298.344,Z 1109.676,A -85,B 0,C 180,E1 14099.908,E2 14099.908} C_VEL
LIN {X 0,Y 296.832,Z 1101.491,A -85,B 0,C 180,E1 14096.142,E2 14096.142} C_VEL
LIN {X 0,Y 297.716,Z 1098.416,A -85,B 0,C 180,E1 14095.015,E2 14095.015} C_VEL
LIN {X 0,Y 303.943,Z 1086.007,A -85,B 0,C 180,E1 14091.316,E2 14091.316} C_VEL
LIN {X 0,Y 311.092,Z 1071.908,A -85,B 0,C 180,E1 14087.799,E2 14087.799} C_VEL
LIN {X 0,Y 318.317,Z 1057.201,A -85,B 0,C 180,E1 14084.775,E2 14084.775} C_VEL
LIN {X 0,Y 326.551,Z 1039.732,A -85,B 0,C 180,E1 14081.789,E2 14081.789} C_VEL
LIN {X 0,Y 333.67,Z 1023.646,A -85,B 0,C 180,E1 14079.501,E2 14079.501} C_VEL
LIN {X 0,Y 341.522,Z 1004.345,A -85,B 0,C 180,E1 14077.22,E2 14077.22} C_VEL
LIN {X 0,Y 348.686,Z 985.039,A -85,B 0,C 180,E1 14075.333,E2 14075.333} C_VEL
LIN {X 0,Y 355.234,Z 964.821,A -85,B 0,C 180,E1 14073.723,E2 14073.723} C_VEL
LIN {X 0,Y 361.111,Z 944.334,A -85,B 0,C 180,E1 14072.382,E2 14072.382} C_VEL
LIN {X 0,Y 366.266,Z 922.349,A -85,B 0,C 180,E1 14071.244,E2 14071.244} C_VEL
LIN {X 0,Y 370.721,Z 898.908,A -85,B 0,C 180,E1 14070.304,E2 14070.304} C_VEL
LIN {X 0,Y 373.821,Z 876.941,A -85,B 0,C 180,E1 14069.66,E2 14069.66} C_VEL
LIN {X 0,Y 376.494,Z 845.542,A -85,B 0,C 180,E1 14068.993,E2 14068.993} C_VEL
LIN {X 0,Y 388.918,Z 670.019,A -85,B 0,C 180,E1 14065.536,E2 14065.536} C_VEL
LIN {X 0,Y 381.661,Z 658.473,A -85,B 0,C 180,E1 14062.569,E2 14062.569} C_VEL
LIN {X 0,Y 375.278,Z 649.06,A -85,B 0,C 180,E1 14059.535,E2 14059.535} C_VEL
LIN {X 0,Y 371.893,Z 644.291,A -85,B 0,C 180,E1 14057.687,E2 14057.687} C_VEL
LIN {X 0,Y 368.603,Z 639.682,A -85,B 0,C 180,E1 14055.651,E2 14055.651} C_VEL
LIN {X 0,Y 365.357,Z 635.041,A -85,B 0,C 180,E1 14053.29,E2 14053.29} C_VEL
LIN {X 0,Y 362.379,Z 631.057,A -85,B 0,C 180,E1 14050.653,E2 14050.653} C_VEL
LIN {X 0,Y 361.654,Z 629.856,A -85,B 0,C 180,E1 14049.87,E2 14049.87} C_VEL
LIN {X 0,Y 358.738,Z 626.443,A -85,B 0,C 180,E1 14045.919,E2 14045.919} C_VEL
LIN {X 0,Y 357.97,Z 624.128,A -85,B 0,C 180,E1 14043.844,E2 14043.844} C_VEL
LIN {X 0,Y 358.061,Z 624.184,A -85,B 0,C 180,E1 14036.398,E2 14036.398} C_VEL
LIN {X 0,Y 359.784,Z 628.159,A -85,B 0,C 180,E1 14032.816,E2 14032.816} C_VEL
LIN {X 0,Y 362.027,Z 630.299,A -85,B 0,C 180,E1 14030.221,E2 14030.221} C_VEL
LIN {X 0,Y 364.757,Z 634.487,A -85,B 0,C 180,E1 14027.655,E2 14027.655} C_VEL
LIN {X 0,Y 366.151,Z 636.122,A -85,B 0,C 180,E1 14026.579,E2 14026.579} C_VEL
LIN {X 0,Y 369.908,Z 641.423,A -85,B 0,C 180,E1 14023.996,E2 14023.996} C_VEL
LIN {X 0,Y 374.081,Z 647.407,A -85,B 0,C 180,E1 14021.575,E2 14021.575} C_VEL
LIN {X 0,Y 378.118,Z 653.285,A -85,B 0,C 180,E1 14019.531,E2 14019.531} C_VEL
LIN {X 0,Y 385.194,Z 665.302,A -85,B 0,C 180,E1 14016.357,E2 14016.357} C_VEL
LIN {X 0,Y 389.042,Z 672.608,A -85,B 0,C 180,E1 14014.799,E2 14014.799} C_VEL
LIN {X 0,Y 374.569,Z 876.92,A -85,B 0,C 180,E1 14010.776,E2 14010.776} C_VEL
LIN {X 0,Y 372.09,Z 899.534,A -85,B 0,C 180,E1 14010.24,E2 14010.24} C_VEL
LIN {X 0,Y 368.125,Z 922.883,A -85,B 0,C 180,E1 14009.507,E2 14009.507} C_VEL
LIN {X 0,Y 363.468,Z 944.82,A -85,B 0,C 180,E1 14008.59,E2 14008.59} C_VEL
LIN {X 0,Y 357.873,Z 966.062,A -85,B 0,C 180,E1 14007.434,E2 14007.434} C_VEL
LIN {X 0,Y 351.513,Z 987.183,A -85,B 0,C 180,E1 14006.012,E2 14006.012} C_VEL
LIN {X 0,Y 344.581,Z 1007.184,A -85,B 0,C 180,E1 14004.337,E2 14004.337} C_VEL
LIN {X 0,Y 336.582,Z 1028.054,A -85,B 0,C 180,E1 14002.203,E2 14002.203} C_VEL
LIN {X 0,Y 329.085,Z 1046.034,A -85,B 0,C 180,E1 13999.965,E2 13999.965} C_VEL
LIN {X 0,Y 320.973,Z 1064.168,A -85,B 0,C 180,E1 13997.228,E2 13997.228} C_VEL
LIN {X 0,Y 313.461,Z 1080.338,A -85,B 0,C 180,E1 13994.311,E2 13994.311} C_VEL
LIN {X 0,Y 306.193,Z 1095.35,A -85,B 0,C 180,E1 13991.022,E2 13991.022} C_VEL
LIN {X 0,Y 299.577,Z 1109.222,A -85,B 0,C 180,E1 13987.404,E2 13987.404} C_VEL
LIN {X 0,Y 293.764,Z 1121.55,A -85,B 0,C 180,E1 13983.501,E2 13983.501} C_VEL
LIN {X 0,Y 288.625,Z 1133.256,A -85,B 0,C 180,E1 13979.012,E2 13979.012} C_VEL
LIN {X 0,Y 285.015,Z 1142.503,A -85,B 0,C 180,E1 13974.674,E2 13974.674} C_VEL
LIN {X 0,Y 282.423,Z 1150.318,A -85,B 0,C 180,E1 13970.084,E2 13970.084} C_VEL
LIN {X 0,Y 280.929,Z 1156.263,A -85,B 0,C 180,E1 13965.693,E2 13965.693} C_VEL
LIN {X 0,Y 280.187,Z 1160.829,A -85,B 0,C 180,E1 13961.087,E2 13961.087} C_VEL
LIN {X 0,Y 279.972,Z 1163.385,A -85,B 0,C 180,E1 13957.386,E2 13957.386} C_VEL
LIN {X 0,Y 279.956,Z 1165.095,A -85,B 0,C 180,E1 13953.275,E2 13953.275} C_VEL
LIN {X 0,Y 279.972,Z 1165.431,A -85,B 0,C 180,E1 13949.181,E2 13949.181} C_VEL
LIN {X 0,Y 279.97,Z 1164.669,A -85,B 0,C 180,E1 13945.493,E2 13945.493} C_VEL
LIN {X 0,Y 280.032,Z 1162.742,A -85,B 0,C 180,E1 13941.501,E2 13941.501} C_VEL
LIN {X 0,Y 280.438,Z 1158.92,A -85,B 0,C 180,E1 13936.809,E2 13936.809} C_VEL
LIN {X 0,Y 281.406,Z 1154.147,A -85,B 0,C 180,E1 13932.634,E2 13932.634} C_VEL
LIN {X 0,Y 283.449,Z 1146.958,A -85,B 0,C 180,E1 13927.824,E2 13927.824} C_VEL
LIN {X 0,Y 286.244,Z 1139.149,A -85,B 0,C 180,E1 13923.665,E2 13923.665} C_VEL
LIN {X 0,Y 290.537,Z 1128.732,A -85,B 0,C 180,E1 13919.151,E2 13919.151} C_VEL
LIN {X 0,Y 295.64,Z 1117.513,A -85,B 0,C 180,E1 13915.14,E2 13915.14} C_VEL
LIN {X 0,Y 301.877,Z 1104.257,A -85,B 0,C 180,E1 13911.244,E2 13911.244} C_VEL
LIN {X 0,Y 308.917,Z 1089.747,A -85,B 0,C 180,E1 13907.683,E2 13907.683} C_VEL
LIN {X 0,Y 316.095,Z 1074.552,A -85,B 0,C 180,E1 13904.605,E2 13904.605} C_VEL
LIN {X 0,Y 324.023,Z 1057.372,A -85,B 0,C 180,E1 13901.689,E2 13901.689} C_VEL
LIN {X 0,Y 331.391,Z 1040.484,A -85,B 0,C 180,E1 13899.316,E2 13899.316} C_VEL
LIN {X 0,Y 339.668,Z 1020.102,A -85,B 0,C 180,E1 13896.945,E2 13896.945} C_VEL
LIN {X 0,Y 346.359,Z 1002.112,A -85,B 0,C 180,E1 13895.218,E2 13895.218} C_VEL
LIN {X 0,Y 353.358,Z 981.046,A -85,B 0,C 180,E1 13893.558,E2 13893.558} C_VEL
LIN {X 0,Y 359.177,Z 961.204,A -85,B 0,C 180,E1 13892.286,E2 13892.286} C_VEL
LIN {X 0,Y 364.605,Z 939.323,A -85,B 0,C 180,E1 13891.173,E2 13891.173} C_VEL
LIN {X 0,Y 368.758,Z 919.267,A -85,B 0,C 180,E1 13890.373,E2 13890.373} C_VEL
LIN {X 0,Y 372.525,Z 895.382,A -85,B 0,C 180,E1 13889.662,E2 13889.662} C_VEL
LIN {X 0,Y 374.926,Z 871.657,A -85,B 0,C 180,E1 13889.12,E2 13889.12} C_VEL
LIN {X 0,Y 388.954,Z 672.323,A -85,B 0,C 180,E1 13885.203,E2 13885.203} C_VEL
LIN {X 0,Y 382.833,Z 661.378,A -85,B 0,C 180,E1 13882.698,E2 13882.698} C_VEL
LIN {X 0,Y 377.539,Z 652.537,A -85,B 0,C 180,E1 13880.259,E2 13880.259} C_VEL
LIN {X 0,Y 372.686,Z 645.282,A -85,B 0,C 180,E1 13877.728,E2 13877.728} C_VEL
LIN {X 0,Y 368.584,Z 639.662,A -85,B 0,C 180,E1 13875.256,E2 13875.256} C_VEL
LIN {X 0,Y 365.396,Z 635.116,A -85,B 0,C 180,E1 13872.966,E2 13872.966} C_VEL
LIN {X 0,Y 362.283,Z 631.006,A -85,B 0,C 180,E1 13870.254,E2 13870.254} C_VEL
LIN {X 0,Y 361.477,Z 629.687,A -85,B 0,C 180,E1 13869.392,E2 13869.392} C_VEL
LIN {X 0,Y 358.552,Z 626.181,A -85,B 0,C 180,E1 13865.44,E2 13865.44} C_VEL
LIN {X 0,Y 357.875,Z 624.119,A -85,B 0,C 180,E1 13863.684,E2 13863.684} C_VEL
LIN {X 0,Y 357.598,Z 624.035,A -85,B 0,C 180,E1 13856.473,E2 13856.473} C_VEL
LIN {X 0,Y 358.011,Z 624.449,A -85,B 0,C 180,E1 13855.354,E2 13855.354} C_VEL
LIN {X 0,Y 359.885,Z 628.29,A -85,B 0,C 180,E1 13851.854,E2 13851.854} C_VEL
LIN {X 0,Y 361.911,Z 630.216,A -85,B 0,C 180,E1 13849.582,E2 13849.582} C_VEL
LIN {X 0,Y 364.68,Z 634.439,A -85,B 0,C 180,E1 13847.007,E2 13847.007} C_VEL
LIN {X 0,Y 366.082,Z 636.123,A -85,B 0,C 180,E1 13845.931,E2 13845.931} C_VEL
LIN {X 0,Y 369.99,Z 641.653,A -85,B 0,C 180,E1 13843.273,E2 13843.273} C_VEL
LIN {X 0,Y 373.873,Z 647.15,A -85,B 0,C 180,E1 13841.038,E2 13841.038} C_VEL
LIN {X 0,Y 379.305,Z 654.984,A -85,B 0,C 180,E1 13838.343,E2 13838.343} C_VEL
LIN {X 0,Y 385.803,Z 665.142,A -85,B 0,C 180,E1 13835.543,E2 13835.543} C_VEL
LIN {X 0,Y 388.832,Z 670.15,A -85,B 0,C 180,E1 13834.354,E2 13834.354} C_VEL
LIN {X 0,Y 374.97,Z 864.624,A -85,B 0,C 180,E1 13830.522,E2 13830.522} C_VEL
LIN {X 0,Y 372.393,Z 887.815,A -85,B 0,C 180,E1 13829.948,E2 13829.948} C_VEL
LIN {X 0,Y 368.772,Z 909.505,A -85,B 0,C 180,E1 13829.199,E2 13829.199} C_VEL
LIN {X 0,Y 364.22,Z 931.438,A -85,B 0,C 180,E1 13828.218,E2 13828.218} C_VEL
LIN {X 0,Y 359.135,Z 951.176,A -85,B 0,C 180,E1 13827.093,E2 13827.093} C_VEL
LIN {X 0,Y 353.02,Z 971.893,A -85,B 0,C 180,E1 13825.652,E2 13825.652} C_VEL
LIN {X 0,Y 346.242,Z 991.595,A -85,B 0,C 180,E1 13823.957,E2 13823.957} C_VEL
LIN {X 0,Y 338.746,Z 1011.282,A -85,B 0,C 180,E1 13821.91,E2 13821.91} C_VEL
LIN {X 0,Y 331.49,Z 1028.536,A -85,B 0,C 180,E1 13819.74,E2 13819.74} C_VEL
LIN {X 0,Y 323.069,Z 1047.109,A -85,B 0,C 180,E1 13816.92,E2 13816.92} C_VEL
LIN {X 0,Y 315.402,Z 1063.182,A -85,B 0,C 180,E1 13813.969,E2 13813.969} C_VEL
LIN {X 0,Y 308.094,Z 1077.736,A -85,B 0,C 180,E1 13810.717,E2 13810.717} C_VEL
LIN {X 0,Y 301.348,Z 1091.132,A -85,B 0,C 180,E1 13807.148,E2 13807.148} C_VEL
LIN {X 0,Y 295.305,Z 1103.104,A -85,B 0,C 180,E1 13803.247,E2 13803.247} C_VEL
LIN {X 0,Y 289.999,Z 1114.155,A -85,B 0,C 180,E1 13798.862,E2 13798.862} C_VEL
LIN {X 0,Y 286.127,Z 1122.929,A -85,B 0,C 180,E1 13794.573,E2 13794.573} C_VEL
LIN {X 0,Y 283.241,Z 1130.313,A -85,B 0,C 180,E1 13790.025,E2 13790.025} C_VEL
LIN {X 0,Y 281.488,Z 1135.892,A -85,B 0,C 180,E1 13785.662,E2 13785.662} C_VEL
LIN {X 0,Y 280.487,Z 1140.137,A -85,B 0,C 180,E1 13781.099,E2 13781.099} C_VEL
LIN {X 0,Y 280.111,Z 1142.636,A -85,B 0,C 180,E1 13777.177,E2 13777.177} C_VEL
LIN {X 0,Y 279.99,Z 1144.215,A -85,B 0,C 180,E1 13772.866,E2 13772.866} C_VEL
LIN {X 0,Y 279.981,Z 1144.396,A -85,B 0,C 180,E1 13768.773,E2 13768.773} C_VEL
LIN {X 0,Y 280.036,Z 1143.557,A -85,B 0,C 180,E1 13764.879,E2 13764.879} C_VEL
LIN {X 0,Y 280.321,Z 1141.289,A -85,B 0,C 180,E1 13760.35,E2 13760.35} C_VEL
LIN {X 0,Y 280.97,Z 1137.881,A -85,B 0,C 180,E1 13756.207,E2 13756.207} C_VEL
LIN {X 0,Y 282.485,Z 1132.682,A -85,B 0,C 180,E1 13751.549,E2 13751.549} C_VEL
LIN {X 0,Y 284.882,Z 1125.954,A -85,B 0,C 180,E1 13747.072,E2 13747.072} C_VEL
LIN {X 0,Y 288.53,Z 1117.411,A -85,B 0,C 180,E1 13742.515,E2 13742.515} C_VEL
LIN {X 0,Y 293.138,Z 1107.576,A -85,B 0,C 180,E1 13738.314,E2 13738.314} C_VEL
LIN {X 0,Y 297.716,Z 1098.416,A -85,B 0,C 180,E1 13735.015,E2 13735.015} C_VEL
LIN {X 0,Y 298.756,Z 1094.79,A -85,B 0,C 180,E1 13733.71,E2 13733.71} C_VEL
LIN {X 0,Y 298.709,Z 1085.768,A -85,B 0,C 180,E1 13730.256,E2 13730.256} C_VEL
LIN {X 0,Y 300.093,Z 1081.581,A -85,B 0,C 180,E1 13729.033,E2 13729.033} C_VEL
LIN {X 0,Y 307.605,Z 1067.224,A -85,B 0,C 180,E1 13725.665,E2 13725.665} C_VEL
LIN {X 0,Y 316.139,Z 1050.348,A -85,B 0,C 180,E1 13722.397,E2 13722.397} C_VEL
LIN {X 0,Y 323.981,Z 1034.023,A -85,B 0,C 180,E1 13719.785,E2 13719.785} C_VEL
LIN {X 0,Y 331.839,Z 1016.301,A -85,B 0,C 180,E1 13717.444,E2 13717.444} C_VEL
LIN {X 0,Y 339.601,Z 997.368,A -85,B 0,C 180,E1 13715.359,E2 13715.359} C_VEL
LIN {X 0,Y 346.475,Z 978.345,A -85,B 0,C 180,E1 13713.647,E2 13713.647} C_VEL
LIN {X 0,Y 353.046,Z 958.11,A -85,B 0,C 180,E1 13712.135,E2 13712.135} C_VEL
LIN {X 0,Y 358.471,Z 938.259,A -85,B 0,C 180,E1 13710.942,E2 13710.942} C_VEL
LIN {X 0,Y 363.382,Z 917.311,A -85,B 0,C 180,E1 13709.919,E2 13709.919} C_VEL
LIN {X 0,Y 367.399,Z 895.117,A -85,B 0,C 180,E1 13709.092,E2 13709.092} C_VEL
LIN {X 0,Y 370.574,Z 871.812,A -85,B 0,C 180,E1 13708.452,E2 13708.452} C_VEL
LIN {X 0,Y 376.788,Z 788.872,A -85,B 0,C 180,E1 13706.797,E2 13706.797} C_VEL
LIN {X 0,Y 385.174,Z 674.739,A -85,B 0,C 180,E1 13704.541,E2 13704.541} C_VEL
LIN {X 0,Y 378.662,Z 664.342,A -85,B 0,C 180,E1 13701.736,E2 13701.736} C_VEL
LIN {X 0,Y 373.026,Z 655.854,A -85,B 0,C 180,E1 13698.925,E2 13698.925} C_VEL
LIN {X 0,Y 370.013,Z 651.505,A -85,B 0,C 180,E1 13697.211,E2 13697.211} C_VEL
LIN {X 0,Y 367.064,Z 647.251,A -85,B 0,C 180,E1 13695.321,E2 13695.321} C_VEL
LIN {X 0,Y 363.989,Z 642.75,A -85,B 0,C 180,E1 13693.018,E2 13693.018} C_VEL
LIN {X 0,Y 361.094,Z 638.751,A -85,B 0,C 180,E1 13690.369,E2 13690.369} C_VEL
LIN {X 0,Y 360.383,Z 637.637,A -85,B 0,C 180,E1 13689.583,E2 13689.583} C_VEL
LIN {X 0,Y 357.604,Z 634.154,A -85,B 0,C 180,E1 13685.616,E2 13685.616} C_VEL
LIN {X 0,Y 356.937,Z 632.054,A -85,B 0,C 180,E1 13683.694,E2 13683.694} C_VEL
LIN {X 0,Y 357.025,Z 632.098,A -85,B 0,C 180,E1 13676.548,E2 13676.548} C_VEL
LIN {X 0,Y 358.808,Z 636.173,A -85,B 0,C 180,E1 13672.797,E2 13672.797} C_VEL
LIN {X 0,Y 360.819,Z 638.15,A -85,B 0,C 180,E1 13670.43,E2 13670.43} C_VEL
LIN {X 0,Y 363.593,Z 642.383,A -85,B 0,C 180,E1 13667.776,E2 13667.776} C_VEL
LIN {X 0,Y 364.761,Z 643.84,A -85,B 0,C 180,E1 13666.85,E2 13666.85} C_VEL
LIN {X 0,Y 368.438,Z 649.171,A -85,B 0,C 180,E1 13664.254,E2 13664.254} C_VEL
LIN {X 0,Y 372.339,Z 654.869,A -85,B 0,C 180,E1 13661.932,E2 13661.932} C_VEL
LIN {X 0,Y 376.287,Z 660.802,A -85,B 0,C 180,E1 13659.873,E2 13659.873} C_VEL
LIN {X 0,Y 382.979,Z 672.488,A -85,B 0,C 180,E1 13656.783,E2 13656.783} C_VEL
LIN {X 0,Y 385.311,Z 677.203,A -85,B 0,C 180,E1 13655.788,E2 13655.788} C_VEL
LIN {X 0,Y 370.591,Z 877.924,A -85,B 0,C 180,E1 13651.834,E2 13651.834} C_VEL
LIN {X 0,Y 367.862,Z 901.484,A -85,B 0,C 180,E1 13651.27,E2 13651.27} C_VEL
LIN {X 0,Y 363.718,Z 924.482,A -85,B 0,C 180,E1 13650.533,E2 13650.533} C_VEL
LIN {X 0,Y 358.647,Z 947.047,A -85,B 0,C 180,E1 13649.568,E2 13649.568} C_VEL
LIN {X 0,Y 353.137,Z 967.241,A -85,B 0,C 180,E1 13648.456,E2 13648.456} C_VEL
LIN {X 0,Y 346.052,Z 989.603,A -85,B 0,C 180,E1 13646.92,E2 13646.92} C_VEL
LIN {X 0,Y 339.256,Z 1008.518,A -85,B 0,C 180,E1 13645.313,E2 13645.313} C_VEL
LIN {X 0,Y 331.012,Z 1029.097,A -85,B 0,C 180,E1 13643.174,E2 13643.174} C_VEL
LIN {X 0,Y 323.029,Z 1047.541,A -85,B 0,C 180,E1 13640.845,E2 13640.845} C_VEL
LIN {X 0,Y 314.935,Z 1064.769,A -85,B 0,C 180,E1 13638.187,E2 13638.187} C_VEL
LIN {X 0,Y 307.087,Z 1080.909,A -85,B 0,C 180,E1 13635.218,E2 13635.218} C_VEL
LIN {X 0,Y 299.524,Z 1095.822,A -85,B 0,C 180,E1 13631.884,E2 13631.884} C_VEL
LIN {X 0,Y 292.275,Z 1110.205,A -85,B 0,C 180,E1 13628.008,E2 13628.008} C_VEL
LIN {X 0,Y 286.478,Z 1121.922,A -85,B 0,C 180,E1 13624.188,E2 13624.188} C_VEL
LIN {X 0,Y 281.119,Z 1133.414,A -85,B 0,C 180,E1 13619.629,E2 13619.629} C_VEL
LIN {X 0,Y 277.312,Z 1142.608,A -85,B 0,C 180,E1 13615.179,E2 13615.179} C_VEL
LIN {X 0,Y 274.566,Z 1150.321,A -85,B 0,C 180,E1 13610.462,E2 13610.462} C_VEL
LIN {X 0,Y 272.929,Z 1156.472,A -85,B 0,C 180,E1 13605.729,E2 13605.729} C_VEL
LIN {X 0,Y 272.2,Z 1160.672,A -85,B 0,C 180,E1 13601.226,E2 13601.226} C_VEL
LIN {X 0,Y 271.971,Z 1163.32,A -85,B 0,C 180,E1 13597.18,E2 13597.18} C_VEL
LIN {X 0,Y 271.964,Z 1164.892,A -85,B 0,C 180,E1 13592.95,E2 13592.95} C_VEL
LIN {X 0,Y 271.981,Z 1165.108,A -85,B 0,C 180,E1 13588.946,E2 13588.946} C_VEL
LIN {X 0,Y 271.97,Z 1164.266,A -85,B 0,C 180,E1 13585.056,E2 13585.056} C_VEL
LIN {X 0,Y 272.064,Z 1162.127,A -85,B 0,C 180,E1 13580.694,E2 13580.694} C_VEL
LIN {X 0,Y 272.529,Z 1158.399,A -85,B 0,C 180,E1 13576.203,E2 13576.203} C_VEL
LIN {X 0,Y 273.664,Z 1153.435,A -85,B 0,C 180,E1 13571.791,E2 13571.791} C_VEL
LIN {X 0,Y 275.9,Z 1146.281,A -85,B 0,C 180,E1 13566.958,E2 13566.958} C_VEL
LIN {X 0,Y 279.146,Z 1138.001,A -85,B 0,C 180,E1 13562.479,E2 13562.479} C_VEL
LIN {X 0,Y 283.614,Z 1127.889,A -85,B 0,C 180,E1 13558.074,E2 13558.074} C_VEL
LIN {X 0,Y 289.093,Z 1116.61,A -85,B 0,C 180,E1 13553.987,E2 13553.987} C_VEL
LIN {X 0,Y 295.438,Z 1103.83,A -85,B 0,C 180,E1 13550.195,E2 13550.195} C_VEL
LIN {X 0,Y 302.855,Z 1089.259,A -85,B 0,C 180,E1 13546.578,E2 13546.578} C_VEL
LIN {X 0,Y 310.5,Z 1073.796,A -85,B 0,C 180,E1 13543.422,E2 13543.422} C_VEL
LIN {X 0,Y 319.33,Z 1055.371,A -85,B 0,C 180,E1 13540.32,E2 13540.32} C_VEL
LIN {X 0,Y 327.089,Z 1038.223,A -85,B 0,C 180,E1 13537.938,E2 13537.938} C_VEL
LIN {X 0,Y 335.073,Z 1019.047,A -85,B 0,C 180,E1 13535.741,E2 13535.741} C_VEL
LIN {X 0,Y 342.313,Z 1000.164,A -85,B 0,C 180,E1 13533.948,E2 13533.948} C_VEL
LIN {X 0,Y 349.231,Z 979.716,A -85,B 0,C 180,E1 13532.37,E2 13532.37} C_VEL
LIN {X 0,Y 355.446,Z 959.035,A -85,B 0,C 180,E1 13531.067,E2 13531.067} C_VEL
LIN {X 0,Y 360.82,Z 937.524,A -85,B 0,C 180,E1 13530.006,E2 13530.006} C_VEL
LIN {X 0,Y 365.372,Z 915.86,A -85,B 0,C 180,E1 13529.172,E2 13529.172} C_VEL
LIN {X 0,Y 368.916,Z 892.689,A -85,B 0,C 180,E1 13528.515,E2 13528.515} C_VEL
LIN {X 0,Y 371.505,Z 865.25,A -85,B 0,C 180,E1 13527.914,E2 13527.914} C_VEL
LIN {X 0,Y 385.217,Z 676.841,A -85,B 0,C 180,E1 13524.211,E2 13524.211} C_VEL
LIN {X 0,Y 379.637,Z 666.734,A -85,B 0,C 180,E1 13521.799,E2 13521.799} C_VEL
LIN {X 0,Y 374.922,Z 658.778,A -85,B 0,C 180,E1 13519.513,E2 13519.513} C_VEL
LIN {X 0,Y 370.246,Z 651.887,A -85,B 0,C 180,E1 13516.957,E2 13516.957} C_VEL
LIN {X 0,Y 366.911,Z 647.081,A -85,B 0,C 180,E1 13514.842,E2 13514.842} C_VEL
LIN {X 0,Y 363.819,Z 642.637,A -85,B 0,C 180,E1 13512.539,E2 13512.539} C_VEL
LIN {X 0,Y 360.851,Z 638.401,A -85,B 0,C 180,E1 13509.811,E2 13509.811} C_VEL
LIN {X 0,Y 360.204,Z 637.461,A -85,B 0,C 180,E1 13509.103,E2 13509.103} C_VEL
LIN {X 0,Y 357.416,Z 633.887,A -85,B 0,C 180,E1 13505.136,E2 13505.136} C_VEL
LIN {X 0,Y 356.836,Z 632.043,A -85,B 0,C 180,E1 13503.534,E2 13503.534} C_VEL
LIN {X 0,Y 356.681,Z 631.992,A -85,B 0,C 180,E1 13496.303,E2 13496.303} C_VEL
LIN {X 0,Y 356.992,Z 632.468,A -85,B 0,C 180,E1 13495.421,E2 13495.421} C_VEL
LIN {X 0,Y 358.911,Z 636.305,A -85,B 0,C 180,E1 13491.832,E2 13491.832} C_VEL
LIN {X 0,Y 360.707,Z 638.09,A -85,B 0,C 180,E1 13489.781,E2 13489.781} C_VEL
LIN {X 0,Y 363.516,Z 642.336,A -85,B 0,C 180,E1 13487.127,E2 13487.127} C_VEL
LIN {X 0,Y 364.69,Z 643.846,A -85,B 0,C 180,E1 13486.2,E2 13486.2} C_VEL
LIN {X 0,Y 368.4,Z 649.208,A -85,B 0,C 180,E1 13483.604,E2 13483.604} C_VEL
LIN {X 0,Y 372.066,Z 654.514,A -85,B 0,C 180,E1 13481.431,E2 13481.431} C_VEL
LIN {X 0,Y 377.301,Z 662.256,A -85,B 0,C 180,E1 13478.753,E2 13478.753} C_VEL
LIN {X 0,Y 383.495,Z 672.16,A -85,B 0,C 180,E1 13476,E2 13476} C_VEL
LIN {X 0,Y 385.098,Z 674.929,A -85,B 0,C 180,E1 13475.34,E2 13475.34} C_VEL
LIN {X 0,Y 371.011,Z 865.908,A -85,B 0,C 180,E1 13471.576,E2 13471.576} C_VEL
LIN {X 0,Y 368.3,Z 889.054,A -85,B 0,C 180,E1 13470.998,E2 13470.998} C_VEL
LIN {X 0,Y 364.67,Z 910.134,A -85,B 0,C 180,E1 13470.269,E2 13470.269} C_VEL
LIN {X 0,Y 359.921,Z 932.249,A -85,B 0,C 180,E1 13469.279,E2 13469.279} C_VEL
LIN {X 0,Y 354.701,Z 951.905,A -85,B 0,C 180,E1 13468.159,E2 13468.159} C_VEL
LIN {X 0,Y 348.208,Z 973.094,A -85,B 0,C 180,E1 13466.678,E2 13466.678} C_VEL
LIN {X 0,Y 341.527,Z 991.905,A -85,B 0,C 180,E1 13465.059,E2 13465.059} C_VEL
LIN {X 0,Y 333.984,Z 1011.117,A -85,B 0,C 180,E1 13463.067,E2 13463.067} C_VEL
LIN {X 0,Y 326.801,Z 1027.644,A -85,B 0,C 180,E1 13460.999,E2 13460.999} C_VEL
LIN {X 0,Y 318.521,Z 1045.421,A -85,B 0,C 180,E1 13458.341,E2 13458.341} C_VEL
LIN {X 0,Y 310.868,Z 1060.759,A -85,B 0,C 180,E1 13455.565,E2 13455.565} C_VEL
LIN {X 0,Y 302.684,Z 1076.534,A -85,B 0,C 180,E1 13452.112,E2 13452.112} C_VEL
LIN {X 0,Y 295.763,Z 1089.609,A -85,B 0,C 180,E1 13448.655,E2 13448.655} C_VEL
LIN {X 0,Y 289.322,Z 1101.69,A -85,B 0,C 180,E1 13444.766,E2 13444.766} C_VEL
LIN {X 0,Y 283.718,Z 1112.675,A -85,B 0,C 180,E1 13440.496,E2 13440.496} C_VEL
LIN {X 0,Y 279.245,Z 1121.875,A -85,B 0,C 180,E1 13436.008,E2 13436.008} C_VEL
LIN {X 0,Y 275.906,Z 1129.742,A -85,B 0,C 180,E1 13431.248,E2 13431.248} C_VEL
LIN {X 0,Y 273.86,Z 1135.461,A -85,B 0,C 180,E1 13426.764,E2 13426.764} C_VEL
LIN {X 0,Y 272.635,Z 1140.134,A -85,B 0,C 180,E1 13421.852,E2 13421.852} C_VEL
LIN {X 0,Y 272.159,Z 1142.719,A -85,B 0,C 180,E1 13417.813,E2 13417.813} C_VEL
LIN {X 0,Y 272.004,Z 1144.349,A -85,B 0,C 180,E1 13413.583,E2 13413.583} C_VEL
LIN {X 0,Y 271.979,Z 1144.74,A -85,B 0,C 180,E1 13409.158,E2 13409.158} C_VEL
LIN {X 0,Y 272.035,Z 1143.988,A -85,B 0,C 180,E1 13405.151,E2 13405.151} C_VEL
LIN {X 0,Y 272.299,Z 1142.011,A -85,B 0,C 180,E1 13400.703,E2 13400.703} C_VEL
LIN {X 0,Y 273.027,Z 1138.385,A -85,B 0,C 180,E1 13396.014,E2 13396.014} C_VEL
LIN {X 0,Y 274.593,Z 1133.367,A -85,B 0,C 180,E1 13391.312,E2 13391.312} C_VEL
LIN {X 0,Y 277.168,Z 1126.604,A -85,B 0,C 180,E1 13386.621,E2 13386.621} C_VEL
LIN {X 0,Y 280.985,Z 1118.248,A -85,B 0,C 180,E1 13381.985,E2 13381.985} C_VEL
LIN {X 0,Y 285.862,Z 1108.387,A -85,B 0,C 180,E1 13377.646,E2 13377.646} C_VEL
LIN {X 0,Y 292.329,Z 1096.075,A -85,B 0,C 180,E1 13373.234,E2 13373.234} C_VEL
LIN {X 0,Y 299.023,Z 1083.566,A -85,B 0,C 180,E1 13369.558,E2 13369.558} C_VEL
LIN {X 0,Y 300.093,Z 1081.581,A -85,B 0,C 180,E1 13369.033,E2 13369.033} C_VEL
LIN {X 0,Y 301.581,Z 1077.3,A -85,B 0,C 180,E1 13367.832,E2 13367.832} C_VEL
LIN {X 0,Y 303.009,Z 1066.298,A -85,B 0,C 180,E1 13364.398,E2 13364.398} C_VEL
LIN {X 0,Y 304.624,Z 1062.223,A -85,B 0,C 180,E1 13363.455,E2 13363.455} C_VEL
LIN {X 0,Y 312.589,Z 1046.89,A -85,B 0,C 180,E1 13360.631,E2 13360.631} C_VEL
LIN {X 0,Y 321.284,Z 1029.06,A -85,B 0,C 180,E1 13357.916,E2 13357.916} C_VEL
LIN {X 0,Y 328.989,Z 1011.979,A -85,B 0,C 180,E1 13355.761,E2 13355.761} C_VEL
LIN {X 0,Y 336.781,Z 992.875,A -85,B 0,C 180,E1 13353.769,E2 13353.769} C_VEL
LIN {X 0,Y 343.663,Z 974.121,A -85,B 0,C 180,E1 13352.152,E2 13352.152} C_VEL
LIN {X 0,Y 350.438,Z 952.801,A -85,B 0,C 180,E1 13350.658,E2 13350.658} C_VEL
LIN {X 0,Y 356.084,Z 932.167,A -85,B 0,C 180,E1 13349.488,E2 13349.488} C_VEL
LIN {X 0,Y 360.942,Z 910.031,A -85,B 0,C 180,E1 13348.509,E2 13348.509} C_VEL
LIN {X 0,Y 364.751,Z 888.4,A -85,B 0,C 180,E1 13347.774,E2 13347.774} C_VEL
LIN {X 0,Y 367.469,Z 865.242,A -85,B 0,C 180,E1 13347.206,E2 13347.206} C_VEL
LIN {X 0,Y 381.591,Z 679.693,A -85,B 0,C 180,E1 13343.553,E2 13343.553} C_VEL
LIN {X 0,Y 375.239,Z 669.262,A -85,B 0,C 180,E1 13340.634,E2 13340.634} C_VEL
LIN {X 0,Y 369.292,Z 660.163,A -85,B 0,C 180,E1 13337.409,E2 13337.409} C_VEL
LIN {X 0,Y 365.415,Z 654.668,A -85,B 0,C 180,E1 13334.905,E2 13334.905} C_VEL
LIN {X 0,Y 362.628,Z 650.458,A -85,B 0,C 180,E1 13332.743,E2 13332.743} C_VEL
LIN {X 0,Y 359.75,Z 646.299,A -85,B 0,C 180,E1 13330.004,E2 13330.004} C_VEL
LIN {X 0,Y 358.979,Z 645.306,A -85,B 0,C 180,E1 13329.135,E2 13329.135} C_VEL
LIN {X 0,Y 356.415,Z 641.682,A -85,B 0,C 180,E1 13325.151,E2 13325.151} C_VEL
LIN {X 0,Y 355.907,Z 639.98,A -85,B 0,C 180,E1 13323.544,E2 13323.544} C_VEL
LIN {X 0,Y 355.992,Z 640.01,A -85,B 0,C 180,E1 13316.7,E2 13316.7} C_VEL
LIN {X 0,Y 357.72,Z 644.051,A -85,B 0,C 180,E1 13312.936,E2 13312.936} C_VEL
LIN {X 0,Y 359.616,Z 645.996,A -85,B 0,C 180,E1 13310.64,E2 13310.64} C_VEL
LIN {X 0,Y 362.43,Z 650.279,A -85,B 0,C 180,E1 13307.898,E2 13307.898} C_VEL
LIN {X 0,Y 363.662,Z 652.061,A -85,B 0,C 180,E1 13306.89,E2 13306.89} C_VEL
LIN {X 0,Y 366.863,Z 656.723,A -85,B 0,C 180,E1 13304.59,E2 13304.59} C_VEL
LIN {X 0,Y 370.677,Z 662.432,A -85,B 0,C 180,E1 13302.254,E2 13302.254} C_VEL
LIN {X 0,Y 374.399,Z 668.195,A -85,B 0,C 180,E1 13300.256,E2 13300.256} C_VEL
LIN {X 0,Y 380.787,Z 679.669,A -85,B 0,C 180,E1 13297.214,E2 13297.214} C_VEL
LIN {X 0,Y 381.701,Z 681.75,A -85,B 0,C 180,E1 13296.797,E2 13296.797} C_VEL
LIN {X 0,Y 366.743,Z 878.913,A -85,B 0,C 180,E1 13292.915,E2 13292.915} C_VEL
LIN {X 0,Y 363.835,Z 902.514,A -85,B 0,C 180,E1 13292.343,E2 13292.343} C_VEL
LIN {X 0,Y 359.695,Z 924.805,A -85,B 0,C 180,E1 13291.629,E2 13291.629} C_VEL
LIN {X 0,Y 354.419,Z 947.471,A -85,B 0,C 180,E1 13290.66,E2 13290.66} C_VEL
LIN {X 0,Y 348.953,Z 966.942,A -85,B 0,C 180,E1 13289.594,E2 13289.594} C_VEL
LIN {X 0,Y 341.663,Z 989.302,A -85,B 0,C 180,E1 13288.067,E2 13288.067} C_VEL
LIN {X 0,Y 334.656,Z 1008.216,A -85,B 0,C 180,E1 13286.468,E2 13286.468} C_VEL
LIN {X 0,Y 326.134,Z 1028.792,A -85,B 0,C 180,E1 13284.334,E2 13284.334} C_VEL
LIN {X 0,Y 317.841,Z 1047.265,A -85,B 0,C 180,E1 13282,E2 13282} C_VEL
LIN {X 0,Y 309.305,Z 1064.73,A -85,B 0,C 180,E1 13279.292,E2 13279.292} C_VEL
LIN {X 0,Y 300.792,Z 1081.457,A -85,B 0,C 180,E1 13276.164,E2 13276.164} C_VEL
LIN {X 0,Y 293.339,Z 1095.51,A -85,B 0,C 180,E1 13272.977,E2 13272.977} C_VEL
LIN {X 0,Y 285.633,Z 1110.023,A -85,B 0,C 180,E1 13269.004,E2 13269.004} C_VEL
LIN {X 0,Y 279.285,Z 1122.195,A -85,B 0,C 180,E1 13264.946,E2 13264.946} C_VEL
LIN {X 0,Y 273.872,Z 1133.102,A -85,B 0,C 180,E1 13260.495,E2 13260.495} C_VEL
LIN {X 0,Y 269.794,Z 1142.297,A -85,B 0,C 180,E1 13255.932,E2 13255.932} C_VEL
LIN {X 0,Y 266.827,Z 1150.012,A -85,B 0,C 180,E1 13251.083,E2 13251.083} C_VEL
LIN {X 0,Y 265.042,Z 1156.165,A -85,B 0,C 180,E1 13246.21,E2 13246.21} C_VEL
LIN {X 0,Y 264.223,Z 1160.454,A -85,B 0,C 180,E1 13241.455,E2 13241.455} C_VEL
LIN {X 0,Y 263.974,Z 1163.137,A -85,B 0,C 180,E1 13237.18,E2 13237.18} C_VEL
LIN {X 0,Y 263.972,Z 1164.617,A -85,B 0,C 180,E1 13232.822,E2 13232.822} C_VEL
LIN {X 0,Y 263.993,Z 1164.784,A -85,B 0,C 180,E1 13228.697,E2 13228.697} C_VEL
LIN {X 0,Y 263.97,Z 1163.924,A -85,B 0,C 180,E1 13224.784,E2 13224.784} C_VEL
LIN {X 0,Y 264.081,Z 1161.686,A -85,B 0,C 180,E1 13220.19,E2 13220.19} C_VEL
LIN {X 0,Y 264.641,Z 1157.877,A -85,B 0,C 180,E1 13215.56,E2 13215.56} C_VEL
LIN {X 0,Y 265.957,Z 1152.735,A -85,B 0,C 180,E1 13210.908,E2 13210.908} C_VEL
LIN {X 0,Y 268.415,Z 1145.604,A -85,B 0,C 180,E1 13206.044,E2 13206.044} C_VEL
LIN {X 0,Y 271.968,Z 1137.271,A -85,B 0,C 180,E1 13201.449,E2 13201.449} C_VEL
LIN {X 0,Y 276.813,Z 1127.006,A -85,B 0,C 180,E1 13196.928,E2 13196.928} C_VEL
LIN {X 0,Y 282.976,Z 1115.031,A -85,B 0,C 180,E1 13192.573,E2 13192.573} C_VEL
LIN {X 0,Y 289.753,Z 1102.195,A -85,B 0,C 180,E1 13188.769,E2 13188.769} C_VEL
LIN {X 0,Y 298.045,Z 1086.535,A -85,B 0,C 180,E1 13184.939,E2 13184.939} C_VEL
LIN {X 0,Y 306.036,Z 1071.175,A -85,B 0,C 180,E1 13181.848,E2 13181.848} C_VEL
LIN {X 0,Y 314.506,Z 1054.03,A -85,B 0,C 180,E1 13179.01,E2 13179.01} C_VEL
LIN {X 0,Y 322.931,Z 1036.056,A -85,B 0,C 180,E1 13176.537,E2 13176.537} C_VEL
LIN {X 0,Y 331.129,Z 1016.766,A -85,B 0,C 180,E1 13174.378,E2 13174.378} C_VEL
LIN {X 0,Y 339.067,Z 996.36,A -85,B 0,C 180,E1 13172.501,E2 13172.501} C_VEL
LIN {X 0,Y 345.917,Z 976.374,A -85,B 0,C 180,E1 13171.015,E2 13171.015} C_VEL
LIN {X 0,Y 352.669,Z 953.626,A -85,B 0,C 180,E1 13169.66,E2 13169.66} C_VEL
LIN {X 0,Y 357.885,Z 932.752,A -85,B 0,C 180,E1 13168.686,E2 13168.686} C_VEL
LIN {X 0,Y 362.556,Z 909.318,A -85,B 0,C 180,E1 13167.864,E2 13167.864} C_VEL
LIN {X 0,Y 365.994,Z 885.841,A -85,B 0,C 180,E1 13167.243,E2 13167.243} C_VEL
LIN {X 0,Y 370.944,Z 822.24,A -85,B 0,C 180,E1 13165.964,E2 13165.964} C_VEL
LIN {X 0,Y 381.562,Z 681.338,A -85,B 0,C 180,E1 13163.186,E2 13163.186} C_VEL
LIN {X 0,Y 375.284,Z 669.831,A -85,B 0,C 180,E1 13160.264,E2 13160.264} C_VEL
LIN {X 0,Y 371.206,Z 663.295,A -85,B 0,C 180,E1 13158.125,E2 13158.125} C_VEL
LIN {X 0,Y 367.884,Z 658.413,A -85,B 0,C 180,E1 13156.175,E2 13156.175} C_VEL
LIN {X 0,Y 365.258,Z 654.494,A -85,B 0,C 180,E1 13154.424,E2 13154.424} C_VEL
LIN {X 0,Y 362.456,Z 650.339,A -85,B 0,C 180,E1 13152.263,E2 13152.263} C_VEL
LIN {X 0,Y 359.508,Z 645.944,A -85,B 0,C 180,E1 13149.444,E2 13149.444} C_VEL
LIN {X 0,Y 356.164,Z 641.208,A -85,B 0,C 180,E1 13144.508,E2 13144.508} C_VEL
LIN {X 0,Y 355.8,Z 639.965,A -85,B 0,C 180,E1 13143.383,E2 13143.383} C_VEL
LIN {X 0,Y 355.767,Z 639.949,A -85,B 0,C 180,E1 13136.132,E2 13136.132} C_VEL
LIN {X 0,Y 358.315,Z 644.703,A -85,B 0,C 180,E1 13131.333,E2 13131.333} C_VEL
LIN {X 0,Y 359.502,Z 645.942,A -85,B 0,C 180,E1 13129.989,E2 13129.989} C_VEL
LIN {X 0,Y 362.354,Z 650.232,A -85,B 0,C 180,E1 13127.247,E2 13127.247} C_VEL
LIN {X 0,Y 363.689,Z 652.246,A -85,B 0,C 180,E1 13126.161,E2 13126.161} C_VEL
LIN {X 0,Y 366.937,Z 656.951,A -85,B 0,C 180,E1 13123.863,E2 13123.863} C_VEL
LIN {X 0,Y 370.537,Z 662.288,A -85,B 0,C 180,E1 13121.677,E2 13121.677} C_VEL
LIN {X 0,Y 375.685,Z 670.155,A -85,B 0,C 180,E1 13118.984,E2 13118.984} C_VEL
LIN {X 0,Y 381.476,Z 679.608,A -85,B 0,C 180,E1 13116.352,E2 13116.352} C_VEL
LIN {X 0,Y 367.371,Z 865.163,A -85,B 0,C 180,E1 13112.697,E2 13112.697} C_VEL
LIN {X 0,Y 364.66,Z 888.303,A -85,B 0,C 180,E1 13112.13,E2 13112.13} C_VEL
LIN {X 0,Y 360.849,Z 909.986,A -85,B 0,C 180,E1 13111.393,E2 13111.393} C_VEL
LIN {X 0,Y 356.251,Z 931.138,A -85,B 0,C 180,E1 13110.466,E2 13110.466} C_VEL
LIN {X 0,Y 350.464,Z 952.387,A -85,B 0,C 180,E1 13109.268,E2 13109.268} C_VEL
LIN {X 0,Y 343.829,Z 973.404,A -85,B 0,C 180,E1 13107.805,E2 13107.805} C_VEL
LIN {X 0,Y 336.943,Z 992.215,A -85,B 0,C 180,E1 13106.191,E2 13106.191} C_VEL
LIN {X 0,Y 328.922,Z 1011.943,A -85,B 0,C 180,E1 13104.14,E2 13104.14} C_VEL
LIN {X 0,Y 321.507,Z 1028.413,A -85,B 0,C 180,E1 13102.068,E2 13102.068} C_VEL
LIN {X 0,Y 312.608,Z 1046.732,A -85,B 0,C 180,E1 13099.292,E2 13099.292} C_VEL
LIN {X 0,Y 304.69,Z 1061.983,A -85,B 0,C 180,E1 13096.489,E2 13096.489} C_VEL
LIN {X 0,Y 296.186,Z 1077.604,A -85,B 0,C 180,E1 13092.994,E2 13092.994} C_VEL
LIN {X 0,Y 288.703,Z 1091.126,A -85,B 0,C 180,E1 13089.33,E2 13089.33} C_VEL
LIN {X 0,Y 281.939,Z 1103.124,A -85,B 0,C 180,E1 13085.315,E2 13085.315} C_VEL
LIN {X 0,Y 275.998,Z 1114.102,A -85,B 0,C 180,E1 13080.842,E2 13080.842} C_VEL
LIN {X 0,Y 271.579,Z 1122.762,A -85,B 0,C 180,E1 13076.455,E2 13076.455} C_VEL
LIN {X 0,Y 268.008,Z 1130.638,A -85,B 0,C 180,E1 13071.446,E2 13071.446} C_VEL
LIN {X 0,Y 265.893,Z 1136.26,A -85,B 0,C 180,E1 13066.832,E2 13066.832} C_VEL
LIN {X 0,Y 264.629,Z 1140.745,A -85,B 0,C 180,E1 13061.773,E2 13061.773} C_VEL
LIN {X 0,Y 264.152,Z 1143.24,A -85,B 0,C 180,E1 13057.613,E2 13057.613} C_VEL
LIN {X 0,Y 264.002,Z 1144.815,A -85,B 0,C 180,E1 13053.04,E2 13053.04} C_VEL
LIN {X 0,Y 263.994,Z 1144.996,A -85,B 0,C 180,E1 13048.698,E2 13048.698} C_VEL
LIN {X 0,Y 264.053,Z 1144.223,A -85,B 0,C 180,E1 13044.786,E2 13044.786} C_VEL
LIN {X 0,Y 264.36,Z 1142.197,A -85,B 0,C 180,E1 13040.201,E2 13040.201} C_VEL
LIN {X 0,Y 265.199,Z 1138.49,A -85,B 0,C 180,E1 13035.369,E2 13035.369} C_VEL
LIN {X 0,Y 266.942,Z 1133.415,A -85,B 0,C 180,E1 13030.528,E2 13030.528} C_VEL
LIN {X 0,Y 269.784,Z 1126.569,A -85,B 0,C 180,E1 13025.709,E2 13025.709} C_VEL
LIN {X 0,Y 273.936,Z 1118.108,A -85,B 0,C 180,E1 13020.959,E2 13020.959} C_VEL
LIN {X 0,Y 278.901,Z 1108.696,A -85,B 0,C 180,E1 13016.736,E2 13016.736} C_VEL
LIN {X 0,Y 285.738,Z 1096.384,A -85,B 0,C 180,E1 13012.24,E2 13012.24} C_VEL
LIN {X 0,Y 292.781,Z 1083.874,A -85,B 0,C 180,E1 13008.508,E2 13008.508} C_VEL
LIN {X 0,Y 300.403,Z 1070.026,A -85,B 0,C 180,E1 13005.121,E2 13005.121} C_VEL
LIN {X 0,Y 304.624,Z 1062.223,A -85,B 0,C 180,E1 13003.455,E2 13003.455} C_VEL
LIN {X 0,Y 306.483,Z 1057.429,A -85,B 0,C 180,E1 13002.368,E2 13002.368} C_VEL
LIN {X 0,Y 308.989,Z 1044.953,A -85,B 0,C 180,E1 12999.202,E2 12999.202} C_VEL
LIN {X 0,Y 310.808,Z 1040.407,A -85,B 0,C 180,E1 12998.366,E2 12998.366} C_VEL
LIN {X 0,Y 319.221,Z 1023.351,A -85,B 0,C 180,E1 12995.937,E2 12995.937} C_VEL
LIN {X 0,Y 327.632,Z 1004.537,A -85,B 0,C 180,E1 12993.74,E2 12993.74} C_VEL
LIN {X 0,Y 335.534,Z 985.12,A -85,B 0,C 180,E1 12991.868,E2 12991.868} C_VEL
LIN {X 0,Y 342.71,Z 964.712,A -85,B 0,C 180,E1 12990.279,E2 12990.279} C_VEL
LIN {X 0,Y 349.201,Z 943.602,A -85,B 0,C 180,E1 12988.94,E2 12988.94} C_VEL
LIN {X 0,Y 354.455,Z 922.856,A -85,B 0,C 180,E1 12987.895,E2 12987.895} C_VEL
LIN {X 0,Y 359.36,Z 898.762,A -85,B 0,C 180,E1 12986.959,E2 12986.959} C_VEL
LIN {X 0,Y 362.688,Z 876.722,A -85,B 0,C 180,E1 12986.335,E2 12986.335} C_VEL
LIN {X 0,Y 365.674,Z 843.57,A -85,B 0,C 180,E1 12985.644,E2 12985.644} C_VEL
LIN {X 0,Y 378.087,Z 684.559,A -85,B 0,C 180,E1 12982.528,E2 12982.528} C_VEL
LIN {X 0,Y 372.699,Z 675.698,A -85,B 0,C 180,E1 12979.92,E2 12979.92} C_VEL
LIN {X 0,Y 367.549,Z 667.555,A -85,B 0,C 180,E1 12977.004,E2 12977.004} C_VEL
LIN {X 0,Y 363.785,Z 662.08,A -85,B 0,C 180,E1 12974.484,E2 12974.484} C_VEL
LIN {X 0,Y 361.277,Z 658.164,A -85,B 0,C 180,E1 12972.467,E2 12972.467} C_VEL
LIN {X 0,Y 358.421,Z 653.846,A -85,B 0,C 180,E1 12969.636,E2 12969.636} C_VEL
LIN {X 0,Y 355.25,Z 649.205,A -85,B 0,C 180,E1 12964.682,E2 12964.682} C_VEL
LIN {X 0,Y 354.879,Z 647.909,A -85,B 0,C 180,E1 12963.392,E2 12963.392} C_VEL
LIN {X 0,Y 354.979,Z 648.027,A -85,B 0,C 180,E1 12956.771,E2 12956.771} C_VEL
LIN {X 0,Y 356.744,Z 652.062,A -85,B 0,C 180,E1 12952.917,E2 12952.917} C_VEL
LIN {X 0,Y 358.418,Z 653.838,A -85,B 0,C 180,E1 12950.851,E2 12950.851} C_VEL
LIN {X 0,Y 361.27,Z 658.173,A -85,B 0,C 180,E1 12948.02,E2 12948.02} C_VEL
LIN {X 0,Y 365.302,Z 664.274,A -85,B 0,C 180,E1 12944.929,E2 12944.929} C_VEL
LIN {X 0,Y 369.416,Z 670.576,A -85,B 0,C 180,E1 12942.354,E2 12942.354} C_VEL
LIN {X 0,Y 373.588,Z 677.45,A -85,B 0,C 180,E1 12940.089,E2 12940.089} C_VEL
LIN {X 0,Y 378.213,Z 686.268,A -85,B 0,C 180,E1 12937.825,E2 12937.825} C_VEL
LIN {X 0,Y 363.053,Z 879.64,A -85,B 0,C 180,E1 12934.024,E2 12934.024} C_VEL
LIN {X 0,Y 359.872,Z 903.904,A -85,B 0,C 180,E1 12933.429,E2 12933.429} C_VEL
LIN {X 0,Y 355.688,Z 925.688,A -85,B 0,C 180,E1 12932.729,E2 12932.729} C_VEL
LIN {X 0,Y 350.165,Z 948.466,A -85,B 0,C 180,E1 12931.75,E2 12931.75} C_VEL
LIN {X 0,Y 344.22,Z 968.918,A -85,B 0,C 180,E1 12930.623,E2 12930.623} C_VEL
LIN {X 0,Y 337.078,Z 989.908,A -85,B 0,C 180,E1 12929.174,E2 12929.174} C_VEL
LIN {X 0,Y 329.673,Z 1009.246,A -85,B 0,C 180,E1 12927.533,E2 12927.533} C_VEL
LIN {X 0,Y 321.089,Z 1029.16,A -85,B 0,C 180,E1 12925.451,E2 12925.451} C_VEL
LIN {X 0,Y 312.519,Z 1047.55,A -85,B 0,C 180,E1 12923.114,E2 12923.114} C_VEL
LIN {X 0,Y 303.669,Z 1064.934,A -85,B 0,C 180,E1 12920.396,E2 12920.396} C_VEL
LIN {X 0,Y 294.581,Z 1082.005,A -85,B 0,C 180,E1 12917.15,E2 12917.15} C_VEL
LIN {X 0,Y 286.835,Z 1095.982,A -85,B 0,C 180,E1 12913.922,E2 12913.922} C_VEL
LIN {X 0,Y 278.738,Z 1110.441,A -85,B 0,C 180,E1 12909.859,E2 12909.859} C_VEL
LIN {X 0,Y 272.07,Z 1122.61,A -85,B 0,C 180,E1 12905.692,E2 12905.692} C_VEL
LIN {X 0,Y 266.431,Z 1133.296,A -85,B 0,C 180,E1 12901.171,E2 12901.171} C_VEL
LIN {X 0,Y 261.97,Z 1142.768,A -85,B 0,C 180,E1 12896.278,E2 12896.278} C_VEL
LIN {X 0,Y 258.998,Z 1150.024,A -85,B 0,C 180,E1 12891.508,E2 12891.508} C_VEL
LIN {X 0,Y 257.104,Z 1156.078,A -85,B 0,C 180,E1 12886.492,E2 12886.492} C_VEL
LIN {X 0,Y 256.241,Z 1160.271,A -85,B 0,C 180,E1 12881.651,E2 12881.651} C_VEL
LIN {X 0,Y 255.976,Z 1163.071,A -85,B 0,C 180,E1 12876.954,E2 12876.954} C_VEL
LIN {X 0,Y 255.987,Z 1164.366,A -85,B 0,C 180,E1 12872.462,E2 12872.462} C_VEL
LIN {X 0,Y 255.998,Z 1164.484,A -85,B 0,C 180,E1 12868.657,E2 12868.657} C_VEL
LIN {X 0,Y 255.972,Z 1163.623,A -85,B 0,C 180,E1 12864.62,E2 12864.62} C_VEL
LIN {X 0,Y 256.095,Z 1161.382,A -85,B 0,C 180,E1 12859.881,E2 12859.881} C_VEL
LIN {X 0,Y 256.724,Z 1157.57,A -85,B 0,C 180,E1 12855.104,E2 12855.104} C_VEL
LIN {X 0,Y 258.17,Z 1152.425,A -85,B 0,C 180,E1 12850.309,E2 12850.309} C_VEL
LIN {X 0,Y 260.843,Z 1145.276,A -85,B 0,C 180,E1 12845.292,E2 12845.292} C_VEL
LIN {X 0,Y 264.863,Z 1136.523,A -85,B 0,C 180,E1 12840.361,E2 12840.361} C_VEL
LIN {X 0,Y 270.082,Z 1126.202,A -85,B 0,C 180,E1 12835.756,E2 12835.756} C_VEL
LIN {X 0,Y 276.706,Z 1114.06,A -85,B 0,C 180,E1 12831.306,E2 12831.306} C_VEL
LIN {X 0,Y 283.494,Z 1101.878,A -85,B 0,C 180,E1 12827.65,E2 12827.65} C_VEL
LIN {X 0,Y 292.195,Z 1086.219,A -85,B 0,C 180,E1 12823.778,E2 12823.778} C_VEL
LIN {X 0,Y 300.54,Z 1070.859,A -85,B 0,C 180,E1 12820.664,E2 12820.664} C_VEL
LIN {X 0,Y 309.391,Z 1053.617,A -85,B 0,C 180,E1 12817.799,E2 12817.799} C_VEL
LIN {X 0,Y 318.084,Z 1035.72,A -85,B 0,C 180,E1 12815.336,E2 12815.336} C_VEL
LIN {X 0,Y 326.345,Z 1016.937,A -85,B 0,C 180,E1 12813.235,E2 12813.235} C_VEL
LIN {X 0,Y 334.412,Z 996.954,A -85,B 0,C 180,E1 12811.391,E2 12811.391} C_VEL
LIN {X 0,Y 341.446,Z 977.074,A -85,B 0,C 180,E1 12809.912,E2 12809.912} C_VEL
LIN {X 0,Y 348.376,Z 954.606,A -85,B 0,C 180,E1 12808.568,E2 12808.568} C_VEL
LIN {X 0,Y 353.877,Z 933.258,A -85,B 0,C 180,E1 12807.573,E2 12807.573} C_VEL
LIN {X 0,Y 358.794,Z 909.396,A -85,B 0,C 180,E1 12806.738,E2 12806.738} C_VEL
LIN {X 0,Y 362.338,Z 885.916,A -85,B 0,C 180,E1 12806.12,E2 12806.12} C_VEL
LIN {X 0,Y 366.986,Z 828.486,A -85,B 0,C 180,E1 12804.964,E2 12804.964} C_VEL
LIN {X 0,Y 378.042,Z 685.898,A -85,B 0,C 180,E1 12802.149,E2 12802.149} C_VEL
LIN {X 0,Y 371.842,Z 674.516,A -85,B 0,C 180,E1 12799.068,E2 12799.068} C_VEL
LIN {X 0,Y 367.266,Z 667.289,A -85,B 0,C 180,E1 12796.447,E2 12796.447} C_VEL
LIN {X 0,Y 363.733,Z 662.043,A -85,B 0,C 180,E1 12794.08,E2 12794.08} C_VEL
LIN {X 0,Y 361.101,Z 658.042,A -85,B 0,C 180,E1 12791.985,E2 12791.985} C_VEL
LIN {X 0,Y 358.243,Z 653.638,A -85,B 0,C 180,E1 12789.154,E2 12789.154} C_VEL
LIN {X 0,Y 355.115,Z 649.104,A -85,B 0,C 180,E1 12784.359,E2 12784.359} C_VEL
LIN {X 0,Y 354.766,Z 647.886,A -85,B 0,C 180,E1 12783.231,E2 12783.231} C_VEL
LIN {X 0,Y 354.837,Z 647.902,A -85,B 0,C 180,E1 12776.01,E2 12776.01} C_VEL
LIN {X 0,Y 356.611,Z 651.928,A -85,B 0,C 180,E1 12772.265,E2 12772.265} C_VEL
LIN {X 0,Y 358.302,Z 653.788,A -85,B 0,C 180,E1 12770.199,E2 12770.199} C_VEL
LIN {X 0,Y 361.193,Z 658.127,A -85,B 0,C 180,E1 12767.368,E2 12767.368} C_VEL
LIN {X 0,Y 365.37,Z 664.503,A -85,B 0,C 180,E1 12764.199,E2 12764.199} C_VEL
LIN {X 0,Y 368.952,Z 669.956,A -85,B 0,C 180,E1 12761.964,E2 12761.964} C_VEL
LIN {X 0,Y 374.15,Z 678.159,A -85,B 0,C 180,E1 12759.18,E2 12759.18} C_VEL
LIN {X 0,Y 377.967,Z 684.694,A -85,B 0,C 180,E1 12757.365,E2 12757.365} C_VEL
LIN {X 0,Y 363.453,Z 868.795,A -85,B 0,C 180,E1 12753.745,E2 12753.745} C_VEL
LIN {X 0,Y 360.143,Z 893.552,A -85,B 0,C 180,E1 12753.103,E2 12753.103} C_VEL
LIN {X 0,Y 356.436,Z 913.522,A -85,B 0,C 180,E1 12752.397,E2 12752.397} C_VEL
LIN {X 0,Y 351.323,Z 935.294,A -85,B 0,C 180,E1 12751.402,E2 12751.402} C_VEL
LIN {X 0,Y 345.89,Z 954.463,A -85,B 0,C 180,E1 12750.304,E2 12750.304} C_VEL
LIN {X 0,Y 338.709,Z 976.111,A -85,B 0,C 180,E1 12748.767,E2 12748.767} C_VEL
LIN {X 0,Y 331.868,Z 994.131,A -85,B 0,C 180,E1 12747.202,E2 12747.202} C_VEL
LIN {X 0,Y 323.244,Z 1014.379,A -85,B 0,C 180,E1 12745.056,E2 12745.056} C_VEL
LIN {X 0,Y 315.059,Z 1031.872,A -85,B 0,C 180,E1 12742.804,E2 12742.804} C_VEL
LIN {X 0,Y 306.249,Z 1049.042,A -85,B 0,C 180,E1 12740.108,E2 12740.108} C_VEL
LIN {X 0,Y 297.621,Z 1064.991,A -85,B 0,C 180,E1 12737.087,E2 12737.087} C_VEL
LIN {X 0,Y 289.327,Z 1079.43,A -85,B 0,C 180,E1 12733.723,E2 12733.723} C_VEL
LIN {X 0,Y 281.197,Z 1093.313,A -85,B 0,C 180,E1 12729.795,E2 12729.795} C_VEL
LIN {X 0,Y 274.582,Z 1104.558,A -85,B 0,C 180,E1 12725.893,E2 12725.893} C_VEL
LIN {X 0,Y 268.28,Z 1115.537,A -85,B 0,C 180,E1 12721.202,E2 12721.202} C_VEL
LIN {X 0,Y 263.447,Z 1124.647,A -85,B 0,C 180,E1 12716.363,E2 12716.363} C_VEL
LIN {X 0,Y 259.982,Z 1131.827,A -85,B 0,C 180,E1 12711.43,E2 12711.43} C_VEL
LIN {X 0,Y 257.769,Z 1137.511,A -85,B 0,C 180,E1 12706.449,E2 12706.449} C_VEL
LIN {X 0,Y 256.622,Z 1141.356,A -85,B 0,C 180,E1 12701.69,E2 12701.69} C_VEL
LIN {X 0,Y 256.14,Z 1143.87,A -85,B 0,C 180,E1 12697.176,E2 12697.176} C_VEL
LIN {X 0,Y 256.009,Z 1145.178,A -85,B 0,C 180,E1 12692.463,E2 12692.463} C_VEL
LIN {X 0,Y 256.005,Z 1145.274,A -85,B 0,C 180,E1 12688.434,E2 12688.434} C_VEL
LIN {X 0,Y 256.076,Z 1144.395,A -85,B 0,C 180,E1 12684.174,E2 12684.174} C_VEL
LIN {X 0,Y 256.466,Z 1142.043,A -85,B 0,C 180,E1 12679.215,E2 12679.215} C_VEL
LIN {X 0,Y 257.396,Z 1138.596,A -85,B 0,C 180,E1 12674.684,E2 12674.684} C_VEL
LIN {X 0,Y 259.452,Z 1133.13,A -85,B 0,C 180,E1 12669.466,E2 12669.466} C_VEL
LIN {X 0,Y 262.473,Z 1126.534,A -85,B 0,C 180,E1 12664.745,E2 12664.745} C_VEL
LIN {X 0,Y 267.216,Z 1117.522,A -85,B 0,C 180,E1 12659.66,E2 12659.66} C_VEL
LIN {X 0,Y 272.614,Z 1107.999,A -85,B 0,C 180,E1 12655.355,E2 12655.355} C_VEL
LIN {X 0,Y 279.593,Z 1096.07,A -85,B 0,C 180,E1 12650.995,E2 12650.995} C_VEL
LIN {X 0,Y 287.493,Z 1082.781,A -85,B 0,C 180,E1 12647.027,E2 12647.027} C_VEL
LIN {X 0,Y 295.555,Z 1068.669,A -85,B 0,C 180,E1 12643.618,E2 12643.618} C_VEL
LIN {X 0,Y 304.518,Z 1052.457,A -85,B 0,C 180,E1 12640.381,E2 12640.381} C_VEL
LIN {X 0,Y 310.808,Z 1040.407,A -85,B 0,C 180,E1 12638.366,E2 12638.366} C_VEL
LIN {X 0,Y 312.882,Z 1035.143,A -85,B 0,C 180,E1 12637.403,E2 12637.403} C_VEL
LIN {X 0,Y 316.099,Z 1021.25,A -85,B 0,C 180,E1 12634.54,E2 12634.54} C_VEL
LIN {X 0,Y 318.028,Z 1016.212,A -85,B 0,C 180,E1 12633.82,E2 12633.82} C_VEL
LIN {X 0,Y 326.404,Z 997.553,A -85,B 0,C 180,E1 12631.795,E2 12631.795} C_VEL
LIN {X 0,Y 333.988,Z 978.288,A -85,B 0,C 180,E1 12630.097,E2 12630.097} C_VEL
LIN {X 0,Y 341.13,Z 957.881,A -85,B 0,C 180,E1 12628.617,E2 12628.617} C_VEL
LIN {X 0,Y 347.053,Z 937.796,A -85,B 0,C 180,E1 12627.449,E2 12627.449} C_VEL
LIN {X 0,Y 352.494,Z 915.855,A -85,B 0,C 180,E1 12626.428,E2 12626.428} C_VEL
LIN {X 0,Y 356.498,Z 895.068,A -85,B 0,C 180,E1 12625.687,E2 12625.687} C_VEL
LIN {X 0,Y 359.892,Z 871.256,A -85,B 0,C 180,E1 12625.059,E2 12625.059} C_VEL
LIN {X 0,Y 374.362,Z 693.876,A -85,B 0,C 180,E1 12621.579,E2 12621.579} C_VEL
LIN {X 0,Y 374.702,Z 689.537,A -85,B 0,C 180,E1 12621.488,E2 12621.488} C_VEL
LIN {X 0,Y 369.679,Z 681.227,A -85,B 0,C 180,E1 12618.898,E2 12618.898} C_VEL
LIN {X 0,Y 365.225,Z 674.137,A -85,B 0,C 180,E1 12616.215,E2 12616.215} C_VEL
LIN {X 0,Y 362.279,Z 669.631,A -85,B 0,C 180,E1 12614.138,E2 12614.138} C_VEL
LIN {X 0,Y 359.934,Z 665.87,A -85,B 0,C 180,E1 12612.188,E2 12612.188} C_VEL
LIN {X 0,Y 356.763,Z 661.065,A -85,B 0,C 180,E1 12608.867,E2 12608.867} C_VEL
LIN {X 0,Y 354.261,Z 657.282,A -85,B 0,C 180,E1 12604.695,E2 12604.695} C_VEL
LIN {X 0,Y 353.853,Z 655.839,A -85,B 0,C 180,E1 12603.24,E2 12603.24} C_VEL
LIN {X 0,Y 353.95,Z 655.933,A -85,B 0,C 180,E1 12596.924,E2 12596.924} C_VEL
LIN {X 0,Y 355.768,Z 660.069,A -85,B 0,C 180,E1 12592.897,E2 12592.897} C_VEL
LIN {X 0,Y 357.225,Z 661.676,A -85,B 0,C 180,E1 12591.064,E2 12591.064} C_VEL
LIN {X 0,Y 360.731,Z 667.143,A -85,B 0,C 180,E1 12587.596,E2 12587.596} C_VEL
LIN {X 0,Y 363.86,Z 672.011,A -85,B 0,C 180,E1 12585.194,E2 12585.194} C_VEL
LIN {X 0,Y 367.643,Z 677.937,A -85,B 0,C 180,E1 12582.756,E2 12582.756} C_VEL
LIN {X 0,Y 371.636,Z 684.747,A -85,B 0,C 180,E1 12580.512,E2 12580.512} C_VEL
LIN {X 0,Y 374.823,Z 691.103,A -85,B 0,C 180,E1 12578.866,E2 12578.866} C_VEL
LIN {X 0,Y 359.489,Z 880.496,A -85,B 0,C 180,E1 12575.152,E2 12575.152} C_VEL
LIN {X 0,Y 355.945,Z 905.829,A -85,B 0,C 180,E1 12574.523,E2 12574.523} C_VEL
LIN {X 0,Y 351.43,Z 928.374,A -85,B 0,C 180,E1 12573.791,E2 12573.791} C_VEL
LIN {X 0,Y 345.705,Z 950.639,A -85,B 0,C 180,E1 12572.809,E2 12572.809} C_VEL
LIN {X 0,Y 339.244,Z 971.954,A -85,B 0,C 180,E1 12571.615,E2 12571.615} C_VEL
LIN {X 0,Y 331.934,Z 992.328,A -85,B 0,C 180,E1 12570.171,E2 12570.171} C_VEL
LIN {X 0,Y 323.563,Z 1013.099,A -85,B 0,C 180,E1 12568.357,E2 12568.357} C_VEL
LIN {X 0,Y 315.342,Z 1031.309,A -85,B 0,C 180,E1 12566.396,E2 12566.396} C_VEL
LIN {X 0,Y 305.542,Z 1051.177,A -85,B 0,C 180,E1 12563.77,E2 12563.77} C_VEL
LIN {X 0,Y 296.532,Z 1068.222,A -85,B 0,C 180,E1 12561.006,E2 12561.006} C_VEL
LIN {X 0,Y 287.465,Z 1084.27,A -85,B 0,C 180,E1 12557.804,E2 12557.804} C_VEL
LIN {X 0,Y 279.085,Z 1098.772,A -85,B 0,C 180,E1 12554.315,E2 12554.315} C_VEL
LIN {X 0,Y 271.328,Z 1111.858,A -85,B 0,C 180,E1 12550.434,E2 12550.434} C_VEL
LIN {X 0,Y 264.009,Z 1124.511,A -85,B 0,C 180,E1 12545.86,E2 12545.86} C_VEL
LIN {X 0,Y 258.571,Z 1134.36,A -85,B 0,C 180,E1 12541.468,E2 12541.468} C_VEL
LIN {X 0,Y 253.799,Z 1143.914,A -85,B 0,C 180,E1 12536.182,E2 12536.182} C_VEL
LIN {X 0,Y 250.838,Z 1150.958,A -85,B 0,C 180,E1 12531.268,E2 12531.268} C_VEL
LIN {X 0,Y 248.983,Z 1156.631,A -85,B 0,C 180,E1 12526.086,E2 12526.086} C_VEL
LIN {X 0,Y 248.211,Z 1160.425,A -85,B 0,C 180,E1 12521.384,E2 12521.384} C_VEL
LIN {X 0,Y 247.987,Z 1163.039,A -85,B 0,C 180,E1 12516.482,E2 12516.482} C_VEL
LIN {X 0,Y 248.001,Z 1164.115,A -85,B 0,C 180,E1 12512.079,E2 12512.079} C_VEL
LIN {X 0,Y 248.004,Z 1164.137,A -85,B 0,C 180,E1 12508.151,E2 12508.151} C_VEL
LIN {X 0,Y 247.982,Z 1163.106,A -85,B 0,C 180,E1 12503.75,E2 12503.75} C_VEL
LIN {X 0,Y 248.185,Z 1160.58,A -85,B 0,C 180,E1 12498.85,E2 12498.85} C_VEL
LIN {X 0,Y 248.925,Z 1156.832,A -85,B 0,C 180,E1 12494.148,E2 12494.148} C_VEL
LIN {X 0,Y 250.75,Z 1151.182,A -85,B 0,C 180,E1 12488.916,E2 12488.916} C_VEL
LIN {X 0,Y 253.678,Z 1144.14,A -85,B 0,C 180,E1 12483.979,E2 12483.979} C_VEL
LIN {X 0,Y 258.327,Z 1134.797,A -85,B 0,C 180,E1 12478.758,E2 12478.758} C_VEL
LIN {X 0,Y 263.796,Z 1124.831,A -85,B 0,C 180,E1 12474.288,E2 12474.288} C_VEL
LIN {X 0,Y 270.951,Z 1112.452,A -85,B 0,C 180,E1 12469.775,E2 12469.775} C_VEL
LIN {X 0,Y 278.722,Z 1099.286,A -85,B 0,C 180,E1 12465.844,E2 12465.844} C_VEL
LIN {X 0,Y 286.964,Z 1085.044,A -85,B 0,C 180,E1 12462.381,E2 12462.381} C_VEL
LIN {X 0,Y 295.961,Z 1069.176,A -85,B 0,C 180,E1 12459.179,E2 12459.179} C_VEL
LIN {X 0,Y 304.898,Z 1052.276,A -85,B 0,C 180,E1 12456.409,E2 12456.409} C_VEL
LIN {X 0,Y 313.976,Z 1034.093,A -85,B 0,C 180,E1 12453.945,E2 12453.945} C_VEL
LIN {X 0,Y 322.562,Z 1015.141,A -85,B 0,C 180,E1 12451.86,E2 12451.86} C_VEL
LIN {X 0,Y 331.237,Z 993.921,A -85,B 0,C 180,E1 12449.964,E2 12449.964} C_VEL
LIN {X 0,Y 338.47,Z 973.858,A -85,B 0,C 180,E1 12448.52,E2 12448.52} C_VEL
LIN {X 0,Y 345.295,Z 951.711,A -85,B 0,C 180,E1 12447.255,E2 12447.255} C_VEL
LIN {X 0,Y 351.184,Z 929.007,A -85,B 0,C 180,E1 12446.241,E2 12446.241} C_VEL
LIN {X 0,Y 355.766,Z 906.185,A -85,B 0,C 180,E1 12445.496,E2 12445.496} C_VEL
LIN {X 0,Y 359.279,Z 881.437,A -85,B 0,C 180,E1 12444.877,E2 12444.877} C_VEL
LIN {X 0,Y 374.188,Z 697.174,A -85,B 0,C 180,E1 12441.258,E2 12441.258} C_VEL
LIN {X 0,Y 374.671,Z 690.751,A -85,B 0,C 180,E1 12441.116,E2 12441.116} C_VEL
LIN {X 0,Y 369.662,Z 681.33,A -85,B 0,C 180,E1 12438.489,E2 12438.489} C_VEL
LIN {X 0,Y 365.301,Z 674.346,A -85,B 0,C 180,E1 12435.885,E2 12435.885} C_VEL
LIN {X 0,Y 362.116,Z 669.45,A -85,B 0,C 180,E1 12433.655,E2 12433.655} C_VEL
LIN {X 0,Y 359.756,Z 665.743,A -85,B 0,C 180,E1 12431.705,E2 12431.705} C_VEL
LIN {X 0,Y 356.716,Z 660.989,A -85,B 0,C 180,E1 12428.543,E2 12428.543} C_VEL
LIN {X 0,Y 354.125,Z 657.187,A -85,B 0,C 180,E1 12424.372,E2 12424.372} C_VEL
LIN {X 0,Y 353.735,Z 655.808,A -85,B 0,C 180,E1 12423.078,E2 12423.078} C_VEL
LIN {X 0,Y 353.806,Z 655.828,A -85,B 0,C 180,E1 12416.151,E2 12416.151} C_VEL
LIN {X 0,Y 355.523,Z 659.807,A -85,B 0,C 180,E1 12412.404,E2 12412.404} C_VEL
LIN {X 0,Y 357.108,Z 661.631,A -85,B 0,C 180,E1 12410.41,E2 12410.41} C_VEL
LIN {X 0,Y 360.564,Z 667,A -85,B 0,C 180,E1 12407.019,E2 12407.019} C_VEL
LIN {X 0,Y 363.925,Z 672.239,A -85,B 0,C 180,E1 12404.462,E2 12404.462} C_VEL
LIN {X 0,Y 367.249,Z 677.418,A -85,B 0,C 180,E1 12402.328,E2 12402.328} C_VEL
LIN {X 0,Y 372.845,Z 686.485,A -85,B 0,C 180,E1 12399.268,E2 12399.268} C_VEL
LIN {X 0,Y 374.579,Z 689.615,A -85,B 0,C 180,E1 12398.406,E2 12398.406} C_VEL
LIN {X 0,Y 359.893,Z 870.056,A -85,B 0,C 180,E1 12394.867,E2 12394.867} C_VEL
LIN {X 0,Y 356.475,Z 894.533,A -85,B 0,C 180,E1 12394.23,E2 12394.23} C_VEL
LIN {X 0,Y 352.593,Z 914.806,A -85,B 0,C 180,E1 12393.514,E2 12393.514} C_VEL
LIN {X 0,Y 347.194,Z 936.882,A -85,B 0,C 180,E1 12392.499,E2 12392.499} C_VEL
LIN {X 0,Y 341.627,Z 955.895,A -85,B 0,C 180,E1 12391.407,E2 12391.407} C_VEL
LIN {X 0,Y 334.48,Z 976.7,A -85,B 0,C 180,E1 12389.93,E2 12389.93} C_VEL
LIN {X 0,Y 327.189,Z 995.325,A -85,B 0,C 180,E1 12388.313,E2 12388.313} C_VEL
LIN {X 0,Y 318.647,Z 1014.689,A -85,B 0,C 180,E1 12386.257,E2 12386.257} C_VEL
LIN {X 0,Y 309.895,Z 1032.784,A -85,B 0,C 180,E1 12383.924,E2 12383.924} C_VEL
LIN {X 0,Y 300.779,Z 1049.853,A -85,B 0,C 180,E1 12381.219,E2 12381.219} C_VEL
LIN {X 0,Y 292.078,Z 1065.303,A -85,B 0,C 180,E1 12378.269,E2 12378.269} C_VEL
LIN {X 0,Y 283.415,Z 1079.742,A -85,B 0,C 180,E1 12374.877,E2 12374.877} C_VEL
LIN {X 0,Y 274.897,Z 1093.626,A -85,B 0,C 180,E1 12370.898,E2 12370.898} C_VEL
LIN {X 0,Y 267.919,Z 1104.871,A -85,B 0,C 180,E1 12366.931,E2 12366.931} C_VEL
LIN {X 0,Y 261.24,Z 1115.849,A -85,B 0,C 180,E1 12362.142,E2 12362.142} C_VEL
LIN {X 0,Y 256.084,Z 1124.958,A -85,B 0,C 180,E1 12357.183,E2 12357.183} C_VEL
LIN {X 0,Y 252.359,Z 1132.136,A -85,B 0,C 180,E1 12352.111,E2 12352.111} C_VEL
LIN {X 0,Y 249.956,Z 1137.818,A -85,B 0,C 180,E1 12346.979,E2 12346.979} C_VEL
LIN {X 0,Y 248.701,Z 1141.66,A -85,B 0,C 180,E1 12342.068,E2 12342.068} C_VEL
LIN {X 0,Y 248.16,Z 1144.172,A -85,B 0,C 180,E1 12337.408,E2 12337.408} C_VEL
LIN {X 0,Y 248.014,Z 1145.478,A -85,B 0,C 180,E1 12332.542,E2 12332.542} C_VEL
LIN {X 0,Y 248.011,Z 1145.574,A -85,B 0,C 180,E1 12328.383,E2 12328.383} C_VEL
LIN {X 0,Y 248.091,Z 1144.695,A -85,B 0,C 180,E1 12323.986,E2 12323.986} C_VEL
LIN {X 0,Y 248.5,Z 1142.46,A -85,B 0,C 180,E1 12319.039,E2 12319.039} C_VEL
LIN {X 0,Y 249.546,Z 1138.901,A -85,B 0,C 180,E1 12314.19,E2 12314.19} C_VEL
LIN {X 0,Y 251.685,Z 1133.675,A -85,B 0,C 180,E1 12309,E2 12309} C_VEL
LIN {X 0,Y 254.859,Z 1127.185,A -85,B 0,C 180,E1 12304.185,E2 12304.185} C_VEL
LIN {X 0,Y 259.609,Z 1118.725,A -85,B 0,C 180,E1 12299.187,E2 12299.187} C_VEL
LIN {X 0,Y 265.525,Z 1108.81,A -85,B 0,C 180,E1 12294.557,E2 12294.557} C_VEL
LIN {X 0,Y 272.827,Z 1097,A -85,B 0,C 180,E1 12290.108,E2 12290.108} C_VEL
LIN {X 0,Y 280.616,Z 1084.488,A -85,B 0,C 180,E1 12286.272,E2 12286.272} C_VEL
LIN {X 0,Y 288.948,Z 1070.639,A -85,B 0,C 180,E1 12282.812,E2 12282.812} C_VEL
LIN {X 0,Y 297.967,Z 1055.152,A -85,B 0,C 180,E1 12279.611,E2 12279.611} C_VEL
LIN {X 0,Y 307.093,Z 1038.221,A -85,B 0,C 180,E1 12276.78,E2 12276.78} C_VEL
LIN {X 0,Y 316.031,Z 1020.508,A -85,B 0,C 180,E1 12274.335,E2 12274.335} C_VEL
LIN {X 0,Y 318.028,Z 1016.212,A -85,B 0,C 180,E1 12273.82,E2 12273.82} C_VEL
LIN {X 0,Y 320.206,Z 1010.466,A -85,B 0,C 180,E1 12272.987,E2 12272.987} C_VEL
LIN {X 0,Y 323.744,Z 995.122,A -85,B 0,C 180,E1 12270.438,E2 12270.438} C_VEL
LIN {X 0,Y 325.547,Z 989.78,A -85,B 0,C 180,E1 12269.82,E2 12269.82} C_VEL
LIN {X 0,Y 333.808,Z 968.297,A -85,B 0,C 180,E1 12268.101,E2 12268.101} C_VEL
LIN {X 0,Y 340.525,Z 948.071,A -85,B 0,C 180,E1 12266.797,E2 12266.797} C_VEL
LIN {X 0,Y 346.638,Z 925.838,A -85,B 0,C 180,E1 12265.659,E2 12265.659} C_VEL
LIN {X 0,Y 351.696,Z 903.273,A -85,B 0,C 180,E1 12264.761,E2 12264.761} C_VEL
LIN {X 0,Y 355.436,Z 880.364,A -85,B 0,C 180,E1 12264.1,E2 12264.1} C_VEL
LIN {X 0,Y 358.403,Z 851.907,A -85,B 0,C 180,E1 12263.492,E2 12263.492} C_VEL
LIN {X 0,Y 371.443,Z 694.533,A -85,B 0,C 180,E1 12260.432,E2 12260.432} C_VEL
LIN {X 0,Y 365.903,Z 685.306,A -85,B 0,C 180,E1 12257.329,E2 12257.329} C_VEL
LIN {X 0,Y 361.615,Z 678.275,A -85,B 0,C 180,E1 12254.41,E2 12254.41} C_VEL
LIN {X 0,Y 358.422,Z 673.381,A -85,B 0,C 180,E1 12251.75,E2 12251.75} C_VEL
LIN {X 0,Y 355.658,Z 668.944,A -85,B 0,C 180,E1 12248.732,E2 12248.732} C_VEL
LIN {X 0,Y 353.219,Z 665.174,A -85,B 0,C 180,E1 12244.546,E2 12244.546} C_VEL
LIN {X 0,Y 352.83,Z 663.769,A -85,B 0,C 180,E1 12243.087,E2 12243.087} C_VEL
LIN {X 0,Y 352.94,Z 663.938,A -85,B 0,C 180,E1 12236.996,E2 12236.996} C_VEL
LIN {X 0,Y 354.793,Z 668.072,A -85,B 0,C 180,E1 12232.877,E2 12232.877} C_VEL
LIN {X 0,Y 356.038,Z 669.511,A -85,B 0,C 180,E1 12231.278,E2 12231.278} C_VEL
LIN {X 0,Y 359.373,Z 674.85,A -85,B 0,C 180,E1 12227.875,E2 12227.875} C_VEL
LIN {X 0,Y 362.427,Z 679.744,A -85,B 0,C 180,E1 12225.461,E2 12225.461} C_VEL
LIN {X 0,Y 366.775,Z 686.629,A -85,B 0,C 180,E1 12222.633,E2 12222.633} C_VEL
LIN {X 0,Y 371.076,Z 694.734,A -85,B 0,C 180,E1 12220.195,E2 12220.195} C_VEL
LIN {X 0,Y 371.557,Z 695.953,A -85,B 0,C 180,E1 12219.926,E2 12219.926} C_VEL
LIN {X 0,Y 356.103,Z 880.997,A -85,B 0,C 180,E1 12216.31,E2 12216.31} C_VEL
LIN {X 0,Y 352.507,Z 905.813,A -85,B 0,C 180,E1 12215.696,E2 12215.696} C_VEL
LIN {X 0,Y 347.892,Z 928.321,A -85,B 0,C 180,E1 12214.974,E2 12214.974} C_VEL
LIN {X 0,Y 342.012,Z 950.585,A -85,B 0,C 180,E1 12214.003,E2 12214.003} C_VEL
LIN {X 0,Y 335.493,Z 971.554,A -85,B 0,C 180,E1 12212.843,E2 12212.843} C_VEL
LIN {X 0,Y 327.887,Z 992.191,A -85,B 0,C 180,E1 12211.396,E2 12211.396} C_VEL
LIN {X 0,Y 319.318,Z 1012.831,A -85,B 0,C 180,E1 12209.607,E2 12209.607} C_VEL
LIN {X 0,Y 310.737,Z 1031.249,A -85,B 0,C 180,E1 12207.634,E2 12207.634} C_VEL
LIN {X 0,Y 300.713,Z 1050.869,A -85,B 0,C 180,E1 12205.045,E2 12205.045} C_VEL
LIN {X 0,Y 291.356,Z 1067.912,A -85,B 0,C 180,E1 12202.28,E2 12202.28} C_VEL
LIN {X 0,Y 281.92,Z 1083.959,A -85,B 0,C 180,E1 12199.062,E2 12199.062} C_VEL
LIN {X 0,Y 273.154,Z 1098.46,A -85,B 0,C 180,E1 12195.543,E2 12195.543} C_VEL
LIN {X 0,Y 264.987,Z 1111.545,A -85,B 0,C 180,E1 12191.612,E2 12191.612} C_VEL
LIN {X 0,Y 257.36,Z 1124.029,A -85,B 0,C 180,E1 12187.026,E2 12187.026} C_VEL
LIN {X 0,Y 251.463,Z 1134.047,A -85,B 0,C 180,E1 12182.465,E2 12182.465} C_VEL
LIN {X 0,Y 246.347,Z 1143.602,A -85,B 0,C 180,E1 12177.038,E2 12177.038} C_VEL
LIN {X 0,Y 243.142,Z 1150.648,A -85,B 0,C 180,E1 12171.975,E2 12171.975} C_VEL
LIN {X 0,Y 241.11,Z 1156.324,A -85,B 0,C 180,E1 12166.626,E2 12166.626} C_VEL
LIN {X 0,Y 240.248,Z 1160.121,A -85,B 0,C 180,E1 12161.766,E2 12161.766} C_VEL
LIN {X 0,Y 239.988,Z 1162.737,A -85,B 0,C 180,E1 12156.699,E2 12156.699} C_VEL
LIN {X 0,Y 240.005,Z 1163.814,A -85,B 0,C 180,E1 12152.148,E2 12152.148} C_VEL
LIN {X 0,Y 240.008,Z 1163.837,A -85,B 0,C 180,E1 12148.09,E2 12148.09} C_VEL
LIN {X 0,Y 239.984,Z 1162.876,A -85,B 0,C 180,E1 12143.781,E2 12143.781} C_VEL
LIN {X 0,Y 240.197,Z 1160.442,A -85,B 0,C 180,E1 12138.717,E2 12138.717} C_VEL
LIN {X 0,Y 240.984,Z 1156.739,A -85,B 0,C 180,E1 12133.859,E2 12133.859} C_VEL
LIN {X 0,Y 242.923,Z 1151.195,A -85,B 0,C 180,E1 12128.465,E2 12128.465} C_VEL
LIN {X 0,Y 246.162,Z 1143.936,A -85,B 0,C 180,E1 12123.2,E2 12123.2} C_VEL
LIN {X 0,Y 251.204,Z 1134.481,A -85,B 0,C 180,E1 12117.767,E2 12117.767} C_VEL
LIN {X 0,Y 257.027,Z 1124.515,A -85,B 0,C 180,E1 12113.196,E2 12113.196} C_VEL
LIN {X 0,Y 264.59,Z 1112.135,A -85,B 0,C 180,E1 12108.599,E2 12108.599} C_VEL
LIN {X 0,Y 272.686,Z 1099.102,A -85,B 0,C 180,E1 12104.655,E2 12104.655} C_VEL
LIN {X 0,Y 281.544,Z 1084.485,A -85,B 0,C 180,E1 12101.07,E2 12101.07} C_VEL
LIN {X 0,Y 290.79,Z 1068.814,A -85,B 0,C 180,E1 12097.896,E2 12097.896} C_VEL
LIN {X 0,Y 300.097,Z 1051.863,A -85,B 0,C 180,E1 12095.118,E2 12095.118} C_VEL
LIN {X 0,Y 309.592,Z 1033.459,A -85,B 0,C 180,E1 12092.638,E2 12092.638} C_VEL
LIN {X 0,Y 318.302,Z 1014.828,A -85,B 0,C 180,E1 12090.604,E2 12090.604} C_VEL
LIN {X 0,Y 327.233,Z 993.609,A -85,B 0,C 180,E1 12088.725,E2 12088.725} C_VEL
LIN {X 0,Y 334.344,Z 974.428,A -85,B 0,C 180,E1 12087.353,E2 12087.353} C_VEL
LIN {X 0,Y 341.29,Z 952.691,A -85,B 0,C 180,E1 12086.11,E2 12086.11} C_VEL
LIN {X 0,Y 346.902,Z 931.817,A -85,B 0,C 180,E1 12085.171,E2 12085.171} C_VEL
LIN {X 0,Y 351.915,Z 908.375,A -85,B 0,C 180,E1 12084.385,E2 12084.385} C_VEL
LIN {X 0,Y 355.578,Z 884.98,A -85,B 0,C 180,E1 12083.784,E2 12083.784} C_VEL
LIN {X 0,Y 360.959,Z 822.027,A -85,B 0,C 180,E1 12082.53,E2 12082.53} C_VEL
LIN {X 0,Y 371.44,Z 695.605,A -85,B 0,C 180,E1 12080.072,E2 12080.072} C_VEL
LIN {X 0,Y 367.136,Z 687.452,A -85,B 0,C 180,E1 12077.677,E2 12077.677} C_VEL
LIN {X 0,Y 363.26,Z 681.213,A -85,B 0,C 180,E1 12075.239,E2 12075.239} C_VEL
LIN {X 0,Y 360.537,Z 676.877,A -85,B 0,C 180,E1 12073.239,E2 12073.239} C_VEL
LIN {X 0,Y 358.419,Z 673.444,A -85,B 0,C 180,E1 12071.423,E2 12071.423} C_VEL
LIN {X 0,Y 355.471,Z 668.755,A -85,B 0,C 180,E1 12068.247,E2 12068.247} C_VEL
LIN {X 0,Y 353.025,Z 664.891,A -85,B 0,C 180,E1 12064.06,E2 12064.06} C_VEL
LIN {X 0,Y 352.706,Z 663.73,A -85,B 0,C 180,E1 12062.925,E2 12062.925} C_VEL
LIN {X 0,Y 352.786,Z 663.785,A -85,B 0,C 180,E1 12056.262,E2 12056.262} C_VEL
LIN {X 0,Y 354.548,Z 667.821,A -85,B 0,C 180,E1 12052.383,E2 12052.383} C_VEL
LIN {X 0,Y 355.919,Z 669.47,A -85,B 0,C 180,E1 12050.622,E2 12050.622} C_VEL
LIN {X 0,Y 359.206,Z 674.713,A -85,B 0,C 180,E1 12047.297,E2 12047.297} C_VEL
LIN {X 0,Y 362.381,Z 679.789,A -85,B 0,C 180,E1 12044.804,E2 12044.804} C_VEL
LIN {X 0,Y 366.638,Z 686.514,A -85,B 0,C 180,E1 12042.051,E2 12042.051} C_VEL
LIN {X 0,Y 371.322,Z 694.487,A -85,B 0,C 180,E1 12039.465,E2 12039.465} C_VEL
LIN {X 0,Y 356.453,Z 871.528,A -85,B 0,C 180,E1 12036.007,E2 12036.007} C_VEL
LIN {X 0,Y 352.974,Z 895.373,A -85,B 0,C 180,E1 12035.384,E2 12035.384} C_VEL
LIN {X 0,Y 348.888,Z 916.089,A -85,B 0,C 180,E1 12034.654,E2 12034.654} C_VEL
LIN {X 0,Y 343.555,Z 937.192,A -85,B 0,C 180,E1 12033.688,E2 12033.688} C_VEL
LIN {X 0,Y 337.494,Z 957.327,A -85,B 0,C 180,E1 12032.537,E2 12032.537} C_VEL
LIN {X 0,Y 330.157,Z 977.902,A -85,B 0,C 180,E1 12031.072,E2 12031.072} C_VEL
LIN {X 0,Y 322.373,Z 997.16,A -85,B 0,C 180,E1 12029.395,E2 12029.395} C_VEL
LIN {X 0,Y 313.976,Z 1015.448,A -85,B 0,C 180,E1 12027.44,E2 12027.44} C_VEL
LIN {X 0,Y 305.151,Z 1033.094,A -85,B 0,C 180,E1 12025.165,E2 12025.165} C_VEL
LIN {X 0,Y 295.997,Z 1049.664,A -85,B 0,C 180,E1 12022.545,E2 12022.545} C_VEL
LIN {X 0,Y 286.667,Z 1065.614,A -85,B 0,C 180,E1 12019.497,E2 12019.497} C_VEL
LIN {X 0,Y 277.624,Z 1080.054,A -85,B 0,C 180,E1 12016.08,E2 12016.08} C_VEL
LIN {X 0,Y 268.703,Z 1093.938,A -85,B 0,C 180,E1 12012.052,E2 12012.052} C_VEL
LIN {X 0,Y 261.258,Z 1105.328,A -85,B 0,C 180,E1 12007.965,E2 12007.965} C_VEL
LIN {X 0,Y 254.235,Z 1116.221,A -85,B 0,C 180,E1 12003.103,E2 12003.103} C_VEL
LIN {X 0,Y 248.776,Z 1125.269,A -85,B 0,C 180,E1 11998.05,E2 11998.05} C_VEL
LIN {X 0,Y 244.769,Z 1132.445,A -85,B 0,C 180,E1 11992.835,E2 11992.835} C_VEL
LIN {X 0,Y 242.134,Z 1138.186,A -85,B 0,C 180,E1 11987.467,E2 11987.467} C_VEL
LIN {X 0,Y 240.739,Z 1142.118,A -85,B 0,C 180,E1 11982.229,E2 11982.229} C_VEL
LIN {X 0,Y 240.16,Z 1144.691,A -85,B 0,C 180,E1 11977.176,E2 11977.176} C_VEL
LIN {X 0,Y 240.02,Z 1145.82,A -85,B 0,C 180,E1 11972.149,E2 11972.149} C_VEL
LIN {X 0,Y 240.019,Z 1145.852,A -85,B 0,C 180,E1 11968.091,E2 11968.091} C_VEL
LIN {X 0,Y 240.12,Z 1144.932,A -85,B 0,C 180,E1 11963.545,E2 11963.545} C_VEL
LIN {X 0,Y 240.591,Z 1142.649,A -85,B 0,C 180,E1 11958.494,E2 11958.494} C_VEL
LIN {X 0,Y 241.709,Z 1139.206,A -85,B 0,C 180,E1 11953.663,E2 11953.663} C_VEL
LIN {X 0,Y 244.014,Z 1134.043,A -85,B 0,C 180,E1 11948.36,E2 11948.36} C_VEL
LIN {X 0,Y 247.61,Z 1127.238,A -85,B 0,C 180,E1 11943.178,E2 11943.178} C_VEL
LIN {X 0,Y 253.073,Z 1118.139,A -85,B 0,C 180,E1 11937.767,E2 11937.767} C_VEL
LIN {X 0,Y 259.163,Z 1108.616,A -85,B 0,C 180,E1 11933.274,E2 11933.274} C_VEL
LIN {X 0,Y 266.929,Z 1096.687,A -85,B 0,C 180,E1 11928.757,E2 11928.757} C_VEL
LIN {X 0,Y 275.63,Z 1083.396,A -85,B 0,C 180,E1 11924.684,E2 11924.684} C_VEL
LIN {X 0,Y 284.428,Z 1069.281,A -85,B 0,C 180,E1 11921.212,E2 11921.212} C_VEL
LIN {X 0,Y 294.145,Z 1053.066,A -85,B 0,C 180,E1 11917.944,E2 11917.944} C_VEL
LIN {X 0,Y 302.87,Z 1037.428,A -85,B 0,C 180,E1 11915.372,E2 11915.372} C_VEL
LIN {X 0,Y 312.768,Z 1018.167,A -85,B 0,C 180,E1 11912.78,E2 11912.78} C_VEL
LIN {X 0,Y 320.889,Z 1000.751,A -85,B 0,C 180,E1 11910.859,E2 11910.859} C_VEL
LIN {X 0,Y 325.547,Z 989.78,A -85,B 0,C 180,E1 11909.82,E2 11909.82} C_VEL
LIN {X 0,Y 327.661,Z 983.489,A -85,B 0,C 180,E1 11909.117,E2 11909.117} C_VEL
LIN {X 0,Y 330.815,Z 967.865,A -85,B 0,C 180,E1 11906.98,E2 11906.98} C_VEL
LIN {X 0,Y 332.744,Z 961.265,A -85,B 0,C 180,E1 11906.366,E2 11906.366} C_VEL
LIN {X 0,Y 339.385,Z 940.299,A -85,B 0,C 180,E1 11905.142,E2 11905.142} C_VEL
LIN {X 0,Y 344.94,Z 919.503,A -85,B 0,C 180,E1 11904.168,E2 11904.168} C_VEL
LIN {X 0,Y 349.536,Z 897.368,A -85,B 0,C 180,E1 11903.374,E2 11903.374} C_VEL
LIN {X 0,Y 353.154,Z 874.267,A -85,B 0,C 180,E1 11902.759,E2 11902.759} C_VEL
LIN {X 0,Y 358.909,Z 809.162,A -85,B 0,C 180,E1 11901.475,E2 11901.475} C_VEL
LIN {X 0,Y 368.264,Z 699.694,A -85,B 0,C 180,E1 11899.344,E2 11899.344} C_VEL
LIN {X 0,Y 363.517,Z 691.575,A -85,B 0,C 180,E1 11896.499,E2 11896.499} C_VEL
LIN {X 0,Y 359.504,Z 685.014,A -85,B 0,C 180,E1 11893.593,E2 11893.593} C_VEL
LIN {X 0,Y 357.101,Z 681.083,A -85,B 0,C 180,E1 11891.467,E2 11891.467} C_VEL
LIN {X 0,Y 354.425,Z 676.711,A -85,B 0,C 180,E1 11888.436,E2 11888.436} C_VEL
LIN {X 0,Y 352.131,Z 672.882,A -85,B 0,C 180,E1 11884.234,E2 11884.234} C_VEL
LIN {X 0,Y 351.81,Z 671.699,A -85,B 0,C 180,E1 11882.933,E2 11882.933} C_VEL
LIN {X 0,Y 351.902,Z 671.737,A -85,B 0,C 180,E1 11877.232,E2 11877.232} C_VEL
LIN {X 0,Y 353.597,Z 675.823,A -85,B 0,C 180,E1 11873.18,E2 11873.18} C_VEL
LIN {X 0,Y 354.798,Z 677.201,A -85,B 0,C 180,E1 11871.574,E2 11871.574} C_VEL
LIN {X 0,Y 358.025,Z 682.554,A -85,B 0,C 180,E1 11868.155,E2 11868.155} C_VEL
LIN {X 0,Y 360.899,Z 687.291,A -85,B 0,C 180,E1 11865.808,E2 11865.808} C_VEL
LIN {X 0,Y 365.012,Z 694.003,A -85,B 0,C 180,E1 11863.039,E2 11863.039} C_VEL
LIN {X 0,Y 368.428,Z 700.73,A -85,B 0,C 180,E1 11861.005,E2 11861.005} C_VEL
LIN {X 0,Y 352.878,Z 881.389,A -85,B 0,C 180,E1 11857.492,E2 11857.492} C_VEL
LIN {X 0,Y 349.216,Z 905.827,A -85,B 0,C 180,E1 11856.891,E2 11856.891} C_VEL
LIN {X 0,Y 344.597,Z 927.855,A -85,B 0,C 180,E1 11856.195,E2 11856.195} C_VEL
LIN {X 0,Y 338.581,Z 950.16,A -85,B 0,C 180,E1 11855.241,E2 11855.241} C_VEL
LIN {X 0,Y 331.684,Z 971.734,A -85,B 0,C 180,E1 11854.061,E2 11854.061} C_VEL
LIN {X 0,Y 324.123,Z 991.727,A -85,B 0,C 180,E1 11852.676,E2 11852.676} C_VEL
LIN {X 0,Y 315.616,Z 1011.751,A -85,B 0,C 180,E1 11850.969,E2 11850.969} C_VEL
LIN {X 0,Y 306.645,Z 1030.46,A -85,B 0,C 180,E1 11848.991,E2 11848.991} C_VEL
LIN {X 0,Y 296.36,Z 1050,A -85,B 0,C 180,E1 11846.442,E2 11846.442} C_VEL
LIN {X 0,Y 287.058,Z 1066.331,A -85,B 0,C 180,E1 11843.82,E2 11843.82} C_VEL
LIN {X 0,Y 277.047,Z 1082.79,A -85,B 0,C 180,E1 11840.563,E2 11840.563} C_VEL
LIN {X 0,Y 267.84,Z 1097.399,A -85,B 0,C 180,E1 11837.027,E2 11837.027} C_VEL
LIN {X 0,Y 259.189,Z 1110.584,A -85,B 0,C 180,E1 11833.063,E2 11833.063} C_VEL
LIN {X 0,Y 251.42,Z 1122.661,A -85,B 0,C 180,E1 11828.635,E2 11828.635} C_VEL
LIN {X 0,Y 244.712,Z 1133.263,A -85,B 0,C 180,E1 11823.757,E2 11823.757} C_VEL
LIN {X 0,Y 239.139,Z 1142.925,A -85,B 0,C 180,E1 11818.194,E2 11818.194} C_VEL
LIN {X 0,Y 235.739,Z 1149.711,A -85,B 0,C 180,E1 11813.231,E2 11813.231} C_VEL
LIN {X 0,Y 233.33,Z 1155.801,A -85,B 0,C 180,E1 11807.455,E2 11807.455} C_VEL
LIN {X 0,Y 232.317,Z 1159.65,A -85,B 0,C 180,E1 11802.426,E2 11802.426} C_VEL
LIN {X 0,Y 231.983,Z 1162.362,A -85,B 0,C 180,E1 11797.18,E2 11797.18} C_VEL
LIN {X 0,Y 232.001,Z 1163.49,A -85,B 0,C 180,E1 11792.47,E2 11792.47} C_VEL
LIN {X 0,Y 232.014,Z 1163.561,A -85,B 0,C 180,E1 11788.271,E2 11788.271} C_VEL
LIN {X 0,Y 231.982,Z 1162.718,A -85,B 0,C 180,E1 11784.062,E2 11784.062} C_VEL
LIN {X 0,Y 232.158,Z 1160.605,A -85,B 0,C 180,E1 11779.076,E2 11779.076} C_VEL
LIN {X 0,Y 232.984,Z 1156.861,A -85,B 0,C 180,E1 11773.802,E2 11773.802} C_VEL
LIN {X 0,Y 234.731,Z 1152.021,A -85,B 0,C 180,E1 11768.772,E2 11768.772} C_VEL
LIN {X 0,Y 238.172,Z 1144.716,A -85,B 0,C 180,E1 11763.038,E2 11763.038} C_VEL
LIN {X 0,Y 242.825,Z 1136.427,A -85,B 0,C 180,E1 11757.914,E2 11757.914} C_VEL
LIN {X 0,Y 249.003,Z 1126.308,A -85,B 0,C 180,E1 11752.963,E2 11752.963} C_VEL
LIN {X 0,Y 256.324,Z 1115.027,A -85,B 0,C 180,E1 11748.46,E2 11748.46} C_VEL
LIN {X 0,Y 264.621,Z 1102.172,A -85,B 0,C 180,E1 11744.347,E2 11744.347} C_VEL
LIN {X 0,Y 273.866,Z 1087.848,A -85,B 0,C 180,E1 11740.589,E2 11740.589} C_VEL
LIN {X 0,Y 283.436,Z 1072.262,A -85,B 0,C 180,E1 11737.298,E2 11737.298} C_VEL
LIN {X 0,Y 293.852,Z 1054.359,A -85,B 0,C 180,E1 11734.224,E2 11734.224} C_VEL
LIN {X 0,Y 302.974,Z 1037.48,A -85,B 0,C 180,E1 11731.871,E2 11731.871} C_VEL
LIN {X 0,Y 312.817,Z 1017.482,A -85,B 0,C 180,E1 11729.61,E2 11729.61} C_VEL
LIN {X 0,Y 321.673,Z 997.607,A -85,B 0,C 180,E1 11727.79,E2 11727.79} C_VEL
LIN {X 0,Y 329.645,Z 976.951,A -85,B 0,C 180,E1 11726.285,E2 11726.285} C_VEL
LIN {X 0,Y 337.046,Z 954.962,A -85,B 0,C 180,E1 11725.003,E2 11725.003} C_VEL
LIN {X 0,Y 343.007,Z 933.562,A -85,B 0,C 180,E1 11724.035,E2 11724.035} C_VEL
LIN {X 0,Y 348.497,Z 908.976,A -85,B 0,C 180,E1 11723.205,E2 11723.205} C_VEL
LIN {X 0,Y 352.256,Z 885.822,A -85,B 0,C 180,E1 11722.613,E2 11722.613} C_VEL
LIN {X 0,Y 356.291,Z 841.488,A -85,B 0,C 180,E1 11721.723,E2 11721.723} C_VEL
LIN {X 0,Y 368.25,Z 700.474,A -85,B 0,C 180,E1 11718.974,E2 11718.974} C_VEL
LIN {X 0,Y 364.745,Z 693.683,A -85,B 0,C 180,E1 11716.892,E2 11716.892} C_VEL
LIN {X 0,Y 359.942,Z 685.653,A -85,B 0,C 180,E1 11713.575,E2 11713.575} C_VEL
LIN {X 0,Y 356.918,Z 680.943,A -85,B 0,C 180,E1 11710.981,E2 11710.981} C_VEL
LIN {X 0,Y 354.235,Z 676.519,A -85,B 0,C 180,E1 11707.949,E2 11707.949} C_VEL
LIN {X 0,Y 351.935,Z 672.594,A -85,B 0,C 180,E1 11703.746,E2 11703.746} C_VEL
LIN {X 0,Y 351.68,Z 671.652,A -85,B 0,C 180,E1 11702.77,E2 11702.77} C_VEL
LIN {X 0,Y 351.758,Z 671.691,A -85,B 0,C 180,E1 11696.414,E2 11696.414} C_VEL
LIN {X 0,Y 353.573,Z 675.832,A -85,B 0,C 180,E1 11692.362,E2 11692.362} C_VEL
LIN {X 0,Y 354.735,Z 677.306,A -85,B 0,C 180,E1 11690.836,E2 11690.836} C_VEL
LIN {X 0,Y 357.857,Z 682.423,A -85,B 0,C 180,E1 11687.576,E2 11687.576} C_VEL
LIN {X 0,Y 360.954,Z 687.52,A -85,B 0,C 180,E1 11685.071,E2 11685.071} C_VEL
LIN {X 0,Y 364.814,Z 693.779,A -85,B 0,C 180,E1 11682.494,E2 11682.494} C_VEL
LIN {X 0,Y 368.154,Z 699.824,A -85,B 0,C 180,E1 11680.535,E2 11680.535} C_VEL
LIN {X 0,Y 353.276,Z 871.851,A -85,B 0,C 180,E1 11677.192,E2 11677.192} C_VEL
LIN {X 0,Y 349.739,Z 895.557,A -85,B 0,C 180,E1 11676.581,E2 11676.581} C_VEL
LIN {X 0,Y 345.6,Z 916.077,A -85,B 0,C 180,E1 11675.868,E2 11675.868} C_VEL
LIN {X 0,Y 340.068,Z 937.502,A -85,B 0,C 180,E1 11674.902,E2 11674.902} C_VEL
LIN {X 0,Y 333.851,Z 957.637,A -85,B 0,C 180,E1 11673.765,E2 11673.765} C_VEL
LIN {X 0,Y 326.32,Z 978.211,A -85,B 0,C 180,E1 11672.316,E2 11672.316} C_VEL
LIN {X 0,Y 318.366,Z 997.353,A -85,B 0,C 180,E1 11670.664,E2 11670.664} C_VEL
LIN {X 0,Y 309.409,Z 1016.276,A -85,B 0,C 180,E1 11668.649,E2 11668.649} C_VEL
LIN {X 0,Y 299.93,Z 1034.559,A -85,B 0,C 180,E1 11666.279,E2 11666.279} C_VEL
LIN {X 0,Y 290.492,Z 1050.975,A -85,B 0,C 180,E1 11663.652,E2 11663.652} C_VEL
LIN {X 0,Y 280.842,Z 1066.757,A -85,B 0,C 180,E1 11660.586,E2 11660.586} C_VEL
LIN {X 0,Y 271.964,Z 1080.367,A -85,B 0,C 180,E1 11657.332,E2 11657.332} C_VEL
LIN {X 0,Y 262.62,Z 1094.25,A -85,B 0,C 180,E1 11653.26,E2 11653.26} C_VEL
LIN {X 0,Y 254.881,Z 1105.495,A -85,B 0,C 180,E1 11649.168,E2 11649.168} C_VEL
LIN {X 0,Y 247.388,Z 1116.472,A -85,B 0,C 180,E1 11644.181,E2 11644.181} C_VEL
LIN {X 0,Y 241.522,Z 1125.579,A -85,B 0,C 180,E1 11638.971,E2 11638.971} C_VEL
LIN {X 0,Y 237.219,Z 1132.754,A -85,B 0,C 180,E1 11633.605,E2 11633.605} C_VEL
LIN {X 0,Y 234.391,Z 1138.431,A -85,B 0,C 180,E1 11628.144,E2 11628.144} C_VEL
LIN {X 0,Y 232.825,Z 1142.422,A -85,B 0,C 180,E1 11622.652,E2 11622.652} C_VEL
LIN {X 0,Y 232.168,Z 1145.075,A -85,B 0,C 180,E1 11617.175,E2 11617.175} C_VEL
LIN {X 0,Y 232.026,Z 1146.121,A -85,B 0,C 180,E1 11612.223,E2 11612.223} C_VEL
LIN {X 0,Y 232.025,Z 1146.152,A -85,B 0,C 180,E1 11608.025,E2 11608.025} C_VEL
LIN {X 0,Y 232.14,Z 1145.233,A -85,B 0,C 180,E1 11603.322,E2 11603.322} C_VEL
LIN {X 0,Y 232.715,Z 1142.798,A -85,B 0,C 180,E1 11597.847,E2 11597.847} C_VEL
LIN {X 0,Y 233.977,Z 1139.312,A -85,B 0,C 180,E1 11592.851,E2 11592.851} C_VEL
LIN {X 0,Y 236.772,Z 1133.622,A -85,B 0,C 180,E1 11587.013,E2 11587.013} C_VEL
LIN {X 0,Y 240.545,Z 1127.116,A -85,B 0,C 180,E1 11581.986,E2 11581.986} C_VEL
LIN {X 0,Y 246.4,Z 1118.001,A -85,B 0,C 180,E1 11576.505,E2 11576.505} C_VEL
LIN {X 0,Y 253.298,Z 1107.92,A -85,B 0,C 180,E1 11571.704,E2 11571.704} C_VEL
LIN {X 0,Y 261.354,Z 1096.14,A -85,B 0,C 180,E1 11567.268,E2 11567.268} C_VEL
LIN {X 0,Y 270.362,Z 1082.947,A -85,B 0,C 180,E1 11563.235,E2 11563.235} C_VEL
LIN {X 0,Y 279.608,Z 1068.756,A -85,B 0,C 180,E1 11559.752,E2 11559.752} C_VEL
LIN {X 0,Y 289.757,Z 1052.37,A -85,B 0,C 180,E1 11556.486,E2 11556.486} C_VEL
LIN {X 0,Y 298.836,Z 1036.634,A -85,B 0,C 180,E1 11553.925,E2 11553.925} C_VEL
LIN {X 0,Y 308.431,Z 1018.468,A -85,B 0,C 180,E1 11551.506,E2 11551.506} C_VEL
LIN {X 0,Y 316.8,Z 1001.051,A -85,B 0,C 180,E1 11549.598,E2 11549.598} C_VEL
LIN {X 0,Y 325.468,Z 980.67,A -85,B 0,C 180,E1 11547.779,E2 11547.779} C_VEL
LIN {X 0,Y 332.744,Z 961.265,A -85,B 0,C 180,E1 11546.366,E2 11546.366} C_VEL
LIN {X 0,Y 334.688,Z 954.569,A -85,B 0,C 180,E1 11545.776,E2 11545.776} C_VEL
LIN {X 0,Y 337.376,Z 937.914,A -85,B 0,C 180,E1 11543.906,E2 11543.906} C_VEL
LIN {X 0,Y 338.848,Z 930.878,A -85,B 0,C 180,E1 11543.416,E2 11543.416} C_VEL
LIN {X 0,Y 344.166,Z 908.939,A -85,B 0,C 180,E1 11542.526,E2 11542.526} C_VEL
LIN {X 0,Y 348.704,Z 884.329,A -85,B 0,C 180,E1 11541.786,E2 11541.786} C_VEL
LIN {X 0,Y 351.578,Z 861.089,A -85,B 0,C 180,E1 11541.271,E2 11541.271} C_VEL
LIN {X 0,Y 365.267,Z 704.943,A -85,B 0,C 180,E1 11538.266,E2 11538.266} C_VEL
LIN {X 0,Y 360.77,Z 697.099,A -85,B 0,C 180,E1 11535.348,E2 11535.348} C_VEL
LIN {X 0,Y 357.656,Z 691.99,A -85,B 0,C 180,E1 11532.924,E2 11532.924} C_VEL
LIN {X 0,Y 355.707,Z 688.684,A -85,B 0,C 180,E1 11531.102,E2 11531.102} C_VEL
LIN {X 0,Y 353.326,Z 684.59,A -85,B 0,C 180,E1 11528.298,E2 11528.298} C_VEL
LIN {X 0,Y 351.096,Z 680.774,A -85,B 0,C 180,E1 11524.083,E2 11524.083} C_VEL
LIN {X 0,Y 350.836,Z 679.64,A -85,B 0,C 180,E1 11522.941,E2 11522.941} C_VEL
LIN {X 0,Y 350.909,Z 679.832,A -85,B 0,C 180,E1 11517.224,E2 11517.224} C_VEL
LIN {X 0,Y 352.731,Z 683.949,A -85,B 0,C 180,E1 11512.999,E2 11512.999} C_VEL
LIN {X 0,Y 353.68,Z 685.174,A -85,B 0,C 180,E1 11511.711,E2 11511.711} C_VEL
LIN {X 0,Y 356.685,Z 690.257,A -85,B 0,C 180,E1 11508.438,E2 11508.438} C_VEL
LIN {X 0,Y 359.484,Z 695.019,A -85,B 0,C 180,E1 11506.079,E2 11506.079} C_VEL
LIN {X 0,Y 363.327,Z 701.493,A -85,B 0,C 180,E1 11503.411,E2 11503.411} C_VEL
LIN {X 0,Y 365.409,Z 705.761,A -85,B 0,C 180,E1 11502.098,E2 11502.098} C_VEL
LIN {X 0,Y 349.821,Z 881.627,A -85,B 0,C 180,E1 11498.699,E2 11498.699} C_VEL
LIN {X 0,Y 346.102,Z 905.719,A -85,B 0,C 180,E1 11498.111,E2 11498.111} C_VEL
LIN {X 0,Y 341.383,Z 927.739,A -85,B 0,C 180,E1 11497.427,E2 11497.427} C_VEL
LIN {X 0,Y 335.272,Z 949.864,A -85,B 0,C 180,E1 11496.496,E2 11496.496} C_VEL
LIN {X 0,Y 328.354,Z 971.059,A -85,B 0,C 180,E1 11495.36,E2 11495.36} C_VEL
LIN {X 0,Y 320.458,Z 991.426,A -85,B 0,C 180,E1 11493.973,E2 11493.973} C_VEL
LIN {X 0,Y 311.69,Z 1011.506,A -85,B 0,C 180,E1 11492.281,E2 11492.281} C_VEL
LIN {X 0,Y 302.58,Z 1029.964,A -85,B 0,C 180,E1 11490.351,E2 11490.351} C_VEL
LIN {X 0,Y 292.192,Z 1049.131,A -85,B 0,C 180,E1 11487.879,E2 11487.879} C_VEL
LIN {X 0,Y 282.502,Z 1065.562,A -85,B 0,C 180,E1 11485.263,E2 11485.263} C_VEL
LIN {X 0,Y 271.812,Z 1082.479,A -85,B 0,C 180,E1 11481.924,E2 11481.924} C_VEL
LIN {X 0,Y 262.201,Z 1097.087,A -85,B 0,C 180,E1 11478.366,E2 11478.366} C_VEL
LIN {X 0,Y 253.126,Z 1110.271,A -85,B 0,C 180,E1 11474.359,E2 11474.359} C_VEL
LIN {X 0,Y 244.916,Z 1122.348,A -85,B 0,C 180,E1 11469.862,E2 11469.862} C_VEL
LIN {X 0,Y 237.787,Z 1132.95,A -85,B 0,C 180,E1 11464.88,E2 11464.88} C_VEL
LIN {X 0,Y 231.807,Z 1142.613,A -85,B 0,C 180,E1 11459.17,E2 11459.17} C_VEL
LIN {X 0,Y 228.127,Z 1149.401,A -85,B 0,C 180,E1 11454.054,E2 11454.054} C_VEL
LIN {X 0,Y 225.5,Z 1155.494,A -85,B 0,C 180,E1 11448.082,E2 11448.082} C_VEL
LIN {X 0,Y 224.368,Z 1159.344,A -85,B 0,C 180,E1 11442.874,E2 11442.874} C_VEL
LIN {X 0,Y 223.989,Z 1162.06,A -85,B 0,C 180,E1 11437.437,E2 11437.437} C_VEL
LIN {X 0,Y 224.003,Z 1163.19,A -85,B 0,C 180,E1 11432.558,E2 11432.558} C_VEL
LIN {X 0,Y 224.019,Z 1163.285,A -85,B 0,C 180,E1 11428.465,E2 11428.465} C_VEL
LIN {X 0,Y 223.985,Z 1162.489,A -85,B 0,C 180,E1 11424.106,E2 11424.106} C_VEL
LIN {X 0,Y 224.146,Z 1160.541,A -85,B 0,C 180,E1 11419.201,E2 11419.201} C_VEL
LIN {X 0,Y 225.05,Z 1156.768,A -85,B 0,C 180,E1 11413.48,E2 11413.48} C_VEL
LIN {X 0,Y 226.911,Z 1151.975,A -85,B 0,C 180,E1 11408.275,E2 11408.275} C_VEL
LIN {X 0,Y 230.771,Z 1144.402,A -85,B 0,C 180,E1 11402.099,E2 11402.099} C_VEL
LIN {X 0,Y 235.773,Z 1136.112,A -85,B 0,C 180,E1 11396.834,E2 11396.834} C_VEL
LIN {X 0,Y 242.355,Z 1125.992,A -85,B 0,C 180,E1 11391.768,E2 11391.768} C_VEL
LIN {X 0,Y 250.1,Z 1114.711,A -85,B 0,C 180,E1 11387.184,E2 11387.184} C_VEL
LIN {X 0,Y 258.704,Z 1102.04,A -85,B 0,C 180,E1 11383.074,E2 11383.074} C_VEL
LIN {X 0,Y 268.504,Z 1087.532,A -85,B 0,C 180,E1 11379.234,E2 11379.234} C_VEL
LIN {X 0,Y 278.43,Z 1071.996,A -85,B 0,C 180,E1 11375.942,E2 11375.942} C_VEL
LIN {X 0,Y 289.266,Z 1054.044,A -85,B 0,C 180,E1 11372.865,E2 11372.865} C_VEL
LIN {X 0,Y 298.809,Z 1036.955,A -85,B 0,C 180,E1 11370.498,E2 11370.498} C_VEL
LIN {X 0,Y 308.841,Z 1017.169,A -85,B 0,C 180,E1 11368.285,E2 11368.285} C_VEL
LIN {X 0,Y 317.827,Z 997.555,A -85,B 0,C 180,E1 11366.508,E2 11366.508} C_VEL
LIN {X 0,Y 326.046,Z 976.841,A -85,B 0,C 180,E1 11365.015,E2 11365.015} C_VEL
LIN {X 0,Y 333.317,Z 955.942,A -85,B 0,C 180,E1 11363.804,E2 11363.804} C_VEL
LIN {X 0,Y 339.554,Z 934.165,A -85,B 0,C 180,E1 11362.827,E2 11362.827} C_VEL
LIN {X 0,Y 345.08,Z 910.361,A -85,B 0,C 180,E1 11362.025,E2 11362.025} C_VEL
LIN {X 0,Y 348.828,Z 888.274,A -85,B 0,C 180,E1 11361.459,E2 11361.459} C_VEL
LIN {X 0,Y 352.102,Z 856.167,A -85,B 0,C 180,E1 11360.801,E2 11360.801} C_VEL
LIN {X 0,Y 365.273,Z 705.438,A -85,B 0,C 180,E1 11357.898,E2 11357.898} C_VEL
LIN {X 0,Y 362.051,Z 699.508,A -85,B 0,C 180,E1 11355.866,E2 11355.866} C_VEL
LIN {X 0,Y 357.956,Z 692.518,A -85,B 0,C 180,E1 11352.83,E2 11352.83} C_VEL
LIN {X 0,Y 355.604,Z 688.64,A -85,B 0,C 180,E1 11350.694,E2 11350.694} C_VEL
LIN {X 0,Y 353.135,Z 684.397,A -85,B 0,C 180,E1 11347.811,E2 11347.811} C_VEL
LIN {X 0,Y 350.899,Z 680.488,A -85,B 0,C 180,E1 11343.594,E2 11343.594} C_VEL
LIN {X 0,Y 350.656,Z 679.574,A -85,B 0,C 180,E1 11342.614,E2 11342.614} C_VEL
LIN {X 0,Y 350.733,Z 679.615,A -85,B 0,C 180,E1 11336.562,E2 11336.562} C_VEL
LIN {X 0,Y 352.488,Z 683.711,A -85,B 0,C 180,E1 11332.502,E2 11332.502} C_VEL
LIN {X 0,Y 353.557,Z 685.139,A -85,B 0,C 180,E1 11331.052,E2 11331.052} C_VEL
LIN {X 0,Y 356.516,Z 690.133,A -85,B 0,C 180,E1 11327.857,E2 11327.857} C_VEL
LIN {X 0,Y 359.536,Z 695.247,A -85,B 0,C 180,E1 11325.341,E2 11325.341} C_VEL
LIN {X 0,Y 363.189,Z 701.389,A -85,B 0,C 180,E1 11322.827,E2 11322.827} C_VEL
LIN {X 0,Y 365.124,Z 705.063,A -85,B 0,C 180,E1 11321.624,E2 11321.624} C_VEL
LIN {X 0,Y 350.252,Z 872.173,A -85,B 0,C 180,E1 11318.398,E2 11318.398} C_VEL
LIN {X 0,Y 346.635,Z 895.871,A -85,B 0,C 180,E1 11317.795,E2 11317.795} C_VEL
LIN {X 0,Y 342.375,Z 916.497,A -85,B 0,C 180,E1 11317.089,E2 11317.089} C_VEL
LIN {X 0,Y 336.736,Z 937.812,A -85,B 0,C 180,E1 11316.141,E2 11316.141} C_VEL
LIN {X 0,Y 330.366,Z 957.947,A -85,B 0,C 180,E1 11315.02,E2 11315.02} C_VEL
